LIN {X 0,Y 291.346,Z 740.192,A -85,B 0,C 180,E1 -16706.302,E2 -16706.302} C_VEL
LIN {X 0,Y 291.388,Z 740.187,A -85,B 0,C 180,E1 -16710.26,E2 -16710.26} C_VEL
LIN {X 0,Y 291.418,Z 740.184,A -85,B 0,C 180,E1 -16714.272,E2 -16714.272} C_VEL
LIN {X 0,Y 291.376,Z 740.187,A -85,B 0,C 180,E1 -16717.299,E2 -16717.299} C_VEL
LIN {X 0,Y 291.459,Z 740.18,A -85,B 0,C 180,E1 -16720.27,E2 -16720.27} C_VEL
LIN {X 0,Y 291.557,Z 740.166,A -85,B 0,C 180,E1 -16724.624,E2 -16724.624} C_VEL
LIN {X 0,Y 291.537,Z 740.167,A -85,B 0,C 180,E1 -16728.881,E2 -16728.881} C_VEL
LIN {X 0,Y 291.689,Z 740.147,A -85,B 0,C 180,E1 -16731.688,E2 -16731.688} C_VEL
LIN {X 0,Y 291.624,Z 740.161,A -85,B 0,C 180,E1 -16734.468,E2 -16734.468} C_VEL
LIN {X 0,Y 291.887,Z 740.128,A -85,B 0,C 180,E1 -16738.62,E2 -16738.62} C_VEL
LIN {X 0,Y 291.887,Z 740.123,A -85,B 0,C 180,E1 -16741.38,E2 -16741.38} C_VEL
LIN {X 0,Y 291.656,Z 740.153,A -85,B 0,C 180,E1 -16746.558,E2 -16746.558} C_VEL
LIN {X 0,Y 291.57,Z 740.163,A -85,B 0,C 180,E1 -16749.714,E2 -16749.714} C_VEL
LIN {X 0,Y 291.517,Z 740.169,A -85,B 0,C 180,E1 -16753.951,E2 -16753.951} C_VEL
LIN {X 0,Y 291.441,Z 740.178,A -85,B 0,C 180,E1 -16758.27,E2 -16758.27} C_VEL
LIN {X 0,Y 291.352,Z 740.195,A -85,B 0,C 180,E1 -16761.213,E2 -16761.213} C_VEL
LIN {X 0,Y 291.329,Z 740.192,A -85,B 0,C 180,E1 -16764.212,E2 -16764.212} C_VEL
LIN {X 0,Y 291.352,Z 740.193,A -85,B 0,C 180,E1 -16767.279,E2 -16767.279} C_VEL
LIN {X 0,Y 291.32,Z 740.194,A -85,B 0,C 180,E1 -16770.439,E2 -16770.439} C_VEL
LIN {X 0,Y 291.345,Z 740.195,A -85,B 0,C 180,E1 -16773.699,E2 -16773.699} C_VEL
LIN {X 0,Y 291.354,Z 740.191,A -85,B 0,C 180,E1 -16777.248,E2 -16777.248} C_VEL
LIN {X 0,Y 291.296,Z 740.2,A -85,B 0,C 180,E1 -16781.589,E2 -16781.589} C_VEL
LIN {X 0,Y 291.283,Z 740.201,A -85,B 0,C 180,E1 -16785.597,E2 -16785.597} C_VEL
LIN {X 0,Y 291.295,Z 740.197,A -85,B 0,C 180,E1 -16789.351,E2 -16789.351} C_VEL
LIN {X 0,Y 291.387,Z 740.185,A -85,B 0,C 180,E1 -16792.916,E2 -16792.916} C_VEL
LIN {X 0,Y 291.345,Z 740.195,A -85,B 0,C 180,E1 -16796.302,E2 -16796.302} C_VEL
LIN {X 0,Y 291.336,Z 740.196,A -85,B 0,C 180,E1 -16800.279,E2 -16800.279} C_VEL
LIN {X 0,Y 291.344,Z 740.195,A -85,B 0,C 180,E1 -16804.265,E2 -16804.265} C_VEL
LIN {X 0,Y 291.353,Z 740.189,A -85,B 0,C 180,E1 -16807.297,E2 -16807.297} C_VEL
LIN {X 0,Y 291.442,Z 740.18,A -85,B 0,C 180,E1 -16810.269,E2 -16810.269} C_VEL
LIN {X 0,Y 291.5,Z 740.176,A -85,B 0,C 180,E1 -16814.665,E2 -16814.665} C_VEL
LIN {X 0,Y 291.53,Z 740.173,A -85,B 0,C 180,E1 -16818.88,E2 -16818.88} C_VEL
LIN {X 0,Y 291.653,Z 740.152,A -85,B 0,C 180,E1 -16821.687,E2 -16821.687} C_VEL
LIN {X 0,Y 291.598,Z 740.16,A -85,B 0,C 180,E1 -16824.468,E2 -16824.468} C_VEL
LIN {X 0,Y 291.879,Z 740.125,A -85,B 0,C 180,E1 -16828.62,E2 -16828.62} C_VEL
LIN {X 0,Y 291.873,Z 740.128,A -85,B 0,C 180,E1 -16831.38,E2 -16831.38} C_VEL
LIN {X 0,Y 291.69,Z 740.149,A -85,B 0,C 180,E1 -16836.919,E2 -16836.919} C_VEL
LIN {X 0,Y 291.571,Z 740.165,A -85,B 0,C 180,E1 -16839.714,E2 -16839.714} C_VEL
LIN {X 0,Y 291.525,Z 740.17,A -85,B 0,C 180,E1 -16843.95,E2 -16843.95} C_VEL
LIN {X 0,Y 291.49,Z 740.173,A -85,B 0,C 180,E1 -16846.818,E2 -16846.818} C_VEL
LIN {X 0,Y 291.454,Z 740.18,A -85,B 0,C 180,E1 -16849.875,E2 -16849.875} C_VEL
LIN {X 0,Y 291.366,Z 740.19,A -85,B 0,C 180,E1 -16854.209,E2 -16854.209} C_VEL
LIN {X 0,Y 291.356,Z 740.19,A -85,B 0,C 180,E1 -16857.279,E2 -16857.279} C_VEL
LIN {X 0,Y 291.321,Z 740.196,A -85,B 0,C 180,E1 -16860.439,E2 -16860.439} C_VEL
LIN {X 0,Y 291.347,Z 740.193,A -85,B 0,C 180,E1 -16863.698,E2 -16863.698} C_VEL
LIN {X 0,Y 291.384,Z 740.186,A -85,B 0,C 180,E1 -16867.255,E2 -16867.255} C_VEL
LIN {X 0,Y 291.399,Z 740.188,A -85,B 0,C 180,E1 -16870.351,E2 -16870.351} C_VEL
LIN {X 0,Y 295.39,Z 753.65,A -85,B 0,C 180,E1 -16871.774,E2 -16871.774} C_VEL
LIN {X 0,Y 298.155,Z 764.257,A -85,B 0,C 180,E1 -16873.124,E2 -16873.124} C_VEL
LIN {X 0,Y 297.198,Z 775.278,A -85,B 0,C 180,E1 -16874.571,E2 -16874.571} C_VEL
LIN {X 0,Y 296.116,Z 785.835,A -85,B 0,C 180,E1 -16876.273,E2 -16876.273} C_VEL
LIN {X 0,Y 294.969,Z 795.249,A -85,B 0,C 180,E1 -16878.153,E2 -16878.153} C_VEL
LIN {X 0,Y 293.97,Z 803.803,A -85,B 0,C 180,E1 -16880.263,E2 -16880.263} C_VEL
LIN {X 0,Y 293.218,Z 810.365,A -85,B 0,C 180,E1 -16882.276,E2 -16882.276} C_VEL
LIN {X 0,Y 292.489,Z 816.762,A -85,B 0,C 180,E1 -16884.782,E2 -16884.782} C_VEL
LIN {X 0,Y 292.073,Z 821.66,A -85,B 0,C 180,E1 -16887.372,E2 -16887.372} C_VEL
LIN {X 0,Y 291.863,Z 825.094,A -85,B 0,C 180,E1 -16890.098,E2 -16890.098} C_VEL
LIN {X 0,Y 292.001,Z 826.918,A -85,B 0,C 180,E1 -16892.787,E2 -16892.787} C_VEL
LIN {X 0,Y 292.268,Z 827.255,A -85,B 0,C 180,E1 -16894.352,E2 -16894.352} C_VEL
LIN {X 0,Y 292.61,Z 827.12,A -85,B 0,C 180,E1 -16895.901,E2 -16895.901} C_VEL
LIN {X 0,Y 293.083,Z 826.429,A -85,B 0,C 180,E1 -16897.438,E2 -16897.438} C_VEL
LIN {X 0,Y 293.687,Z 825.284,A -85,B 0,C 180,E1 -16898.964,E2 -16898.964} C_VEL
LIN {X 0,Y 294.663,Z 822.645,A -85,B 0,C 180,E1 -16901.217,E2 -16901.217} C_VEL
LIN {X 0,Y 296.004,Z 818.763,A -85,B 0,C 180,E1 -16903.446,E2 -16903.446} C_VEL
LIN {X 0,Y 297.717,Z 813.148,A -85,B 0,C 180,E1 -16905.81,E2 -16905.81} C_VEL
LIN {X 0,Y 299.467,Z 806.982,A -85,B 0,C 180,E1 -16907.806,E2 -16907.806} C_VEL
LIN {X 0,Y 301.445,Z 798.721,A -85,B 0,C 180,E1 -16909.929,E2 -16909.929} C_VEL
LIN {X 0,Y 303.384,Z 790.165,A -85,B 0,C 180,E1 -16911.675,E2 -16911.675} C_VEL
LIN {X 0,Y 305.048,Z 781.584,A -85,B 0,C 180,E1 -16913.112,E2 -16913.112} C_VEL
LIN {X 0,Y 305.862,Z 775.886,A -85,B 0,C 180,E1 -16913.953,E2 -16913.953} C_VEL
LIN {X 0,Y 303.788,Z 767.821,A -85,B 0,C 180,E1 -16915.422,E2 -16915.422} C_VEL
LIN {X 0,Y 301.043,Z 760.013,A -85,B 0,C 180,E1 -16916.805,E2 -16916.805} C_VEL
LIN {X 0,Y 295.849,Z 748.049,A -85,B 0,C 180,E1 -16918.837,E2 -16918.837} C_VEL
LIN {X 0,Y 295.454,Z 747.403,A -85,B 0,C 180,E1 -16918.961,E2 -16918.961} C_VEL
LIN {X 0,Y 293.453,Z 745.045,A -85,B 0,C 180,E1 -16919.5,E2 -16919.5} C_VEL
LIN {X 0,Y 289.167,Z 742.472,A -85,B 0,C 180,E1 -16920.454,E2 -16920.454} C_VEL
LIN {X 0,Y 286.173,Z 741.381,A -85,B 0,C 180,E1 -16921.331,E2 -16921.331} C_VEL
LIN {X 0,Y 284.879,Z 741.031,A -85,B 0,C 180,E1 -16922.085,E2 -16922.085} C_VEL
LIN {X 0,Y 284.761,Z 741.007,A -85,B 0,C 180,E1 -16922.352,E2 -16922.352} C_VEL
LIN {X 0,Y 284.689,Z 741.021,A -85,B 0,C 180,E1 -16927.09,E2 -16927.09} C_VEL
LIN {X 0,Y 284.522,Z 741.039,A -85,B 0,C 180,E1 -16929.957,E2 -16929.957} C_VEL
LIN {X 0,Y 284.485,Z 741.043,A -85,B 0,C 180,E1 -16934.303,E2 -16934.303} C_VEL
LIN {X 0,Y 284.428,Z 741.052,A -85,B 0,C 180,E1 -16937.248,E2 -16937.248} C_VEL
LIN {X 0,Y 284.38,Z 741.058,A -85,B 0,C 180,E1 -16940.242,E2 -16940.242} C_VEL
LIN {X 0,Y 284.339,Z 741.065,A -85,B 0,C 180,E1 -16944.846,E2 -16944.846} C_VEL
LIN {X 0,Y 284.33,Z 741.067,A -85,B 0,C 180,E1 -16948.011,E2 -16948.011} C_VEL
LIN {X 0,Y 284.378,Z 741.283,A -85,B 0,C 180,E1 -16949.961,E2 -16949.961} C_VEL
LIN {X 0,Y 284.925,Z 743.801,A -85,B 0,C 180,E1 -16953.002,E2 -16953.002} C_VEL
LIN {X 0,Y 285.653,Z 746.974,A -85,B 0,C 180,E1 -16956.191,E2 -16956.191} C_VEL
LIN {X 0,Y 286.553,Z 750.978,A -85,B 0,C 180,E1 -16959.619,E2 -16959.619} C_VEL
LIN {X 0,Y 287.534,Z 755.832,A -85,B 0,C 180,E1 -16963.187,E2 -16963.187} C_VEL
LIN {X 0,Y 288.642,Z 761.7,A -85,B 0,C 180,E1 -16966.925,E2 -16966.925} C_VEL
LIN {X 0,Y 289.605,Z 767.03,A -85,B 0,C 180,E1 -16969.978,E2 -16969.978} C_VEL
LIN {X 0,Y 289.804,Z 768.763,A -85,B 0,C 180,E1 -16970.911,E2 -16970.911} C_VEL
LIN {X 0,Y 288.885,Z 773.995,A -85,B 0,C 180,E1 -16973.401,E2 -16973.401} C_VEL
LIN {X 0,Y 287.081,Z 782.923,A -85,B 0,C 180,E1 -16977.413,E2 -16977.413} C_VEL
LIN {X 0,Y 286.057,Z 790.173,A -85,B 0,C 180,E1 -16980.457,E2 -16980.457} C_VEL
LIN {X 0,Y 286.958,Z 794.013,A -85,B 0,C 180,E1 -16980.809,E2 -16980.809} C_VEL
LIN {X 0,Y 289.321,Z 804.43,A -85,B 0,C 180,E1 -16981.849,E2 -16981.849} C_VEL
LIN {X 0,Y 291.377,Z 817.452,A -85,B 0,C 180,E1 -16983.181,E2 -16983.181} C_VEL
LIN {X 0,Y 292.203,Z 829.766,A -85,B 0,C 180,E1 -16984.537,E2 -16984.537} C_VEL
LIN {X 0,Y 292.108,Z 840.627,A -85,B 0,C 180,E1 -16985.857,E2 -16985.857} C_VEL
LIN {X 0,Y 291.086,Z 852.313,A -85,B 0,C 180,E1 -16987.462,E2 -16987.462} C_VEL
LIN {X 0,Y 290.017,Z 862.075,A -85,B 0,C 180,E1 -16989.057,E2 -16989.057} C_VEL
LIN {X 0,Y 289.18,Z 867.757,A -85,B 0,C 180,E1 -16990.108,E2 -16990.108} C_VEL
LIN {X 0,Y 286.894,Z 877.547,A -85,B 0,C 180,E1 -16992.169,E2 -16992.169} C_VEL
LIN {X 0,Y 285.252,Z 885.594,A -85,B 0,C 180,E1 -16994.275,E2 -16994.275} C_VEL
LIN {X 0,Y 284.228,Z 892.25,A -85,B 0,C 180,E1 -16996.414,E2 -16996.414} C_VEL
LIN {X 0,Y 283.489,Z 897.677,A -85,B 0,C 180,E1 -16998.561,E2 -16998.561} C_VEL
LIN {X 0,Y 283.215,Z 902.021,A -85,B 0,C 180,E1 -17000.718,E2 -17000.718} C_VEL
LIN {X 0,Y 283.239,Z 905.511,A -85,B 0,C 180,E1 -17002.988,E2 -17002.988} C_VEL
LIN {X 0,Y 283.617,Z 908.327,A -85,B 0,C 180,E1 -17005.737,E2 -17005.737} C_VEL
LIN {X 0,Y 283.773,Z 909.165,A -85,B 0,C 180,E1 -17007.161,E2 -17007.161} C_VEL
LIN {X 0,Y 283.935,Z 909.542,A -85,B 0,C 180,E1 -17008.582,E2 -17008.582} C_VEL
LIN {X 0,Y 284.199,Z 909.518,A -85,B 0,C 180,E1 -17010,E2 -17010} C_VEL
LIN {X 0,Y 284.012,Z 909.006,A -85,B 0,C 180,E1 -17011.418,E2 -17011.418} C_VEL
LIN {X 0,Y 283.895,Z 908.063,A -85,B 0,C 180,E1 -17012.838,E2 -17012.838} C_VEL
LIN {X 0,Y 283.788,Z 906.629,A -85,B 0,C 180,E1 -17014.261,E2 -17014.261} C_VEL
LIN {X 0,Y 283.582,Z 903.606,A -85,B 0,C 180,E1 -17016.403,E2 -17016.403} C_VEL
LIN {X 0,Y 283.483,Z 899.442,A -85,B 0,C 180,E1 -17018.554,E2 -17018.554} C_VEL
LIN {X 0,Y 283.675,Z 893.034,A -85,B 0,C 180,E1 -17021.07,E2 -17021.07} C_VEL
LIN {X 0,Y 284.245,Z 886.007,A -85,B 0,C 180,E1 -17023.221,E2 -17023.221} C_VEL
LIN {X 0,Y 285.215,Z 877.236,A -85,B 0,C 180,E1 -17025.36,E2 -17025.36} C_VEL
LIN {X 0,Y 286.444,Z 867.317,A -85,B 0,C 180,E1 -17027.307,E2 -17027.307} C_VEL
LIN {X 0,Y 287.546,Z 858.519,A -85,B 0,C 180,E1 -17028.711,E2 -17028.711} C_VEL
LIN {X 0,Y 287.331,Z 847.324,A -85,B 0,C 180,E1 -17030.205,E2 -17030.205} C_VEL
LIN {X 0,Y 286.963,Z 834.809,A -85,B 0,C 180,E1 -17031.553,E2 -17031.553} C_VEL
LIN {X 0,Y 286.091,Z 821.64,A -85,B 0,C 180,E1 -17032.667,E2 -17032.667} C_VEL
LIN {X 0,Y 284.91,Z 807.176,A -85,B 0,C 180,E1 -17033.568,E2 -17033.568} C_VEL
LIN {X 0,Y 284.391,Z 801.447,A -85,B 0,C 180,E1 -17033.885,E2 -17033.885} C_VEL
LIN {X 0,Y 285.455,Z 791.716,A -85,B 0,C 180,E1 -17037.891,E2 -17037.891} C_VEL
LIN {X 0,Y 286.689,Z 782.298,A -85,B 0,C 180,E1 -17041.807,E2 -17041.807} C_VEL
LIN {X 0,Y 288.579,Z 771.122,A -85,B 0,C 180,E1 -17046.517,E2 -17046.517} C_VEL
LIN {X 0,Y 289.217,Z 767.266,A -85,B 0,C 180,E1 -17048.16,E2 -17048.16} C_VEL
LIN {X 0,Y 288.67,Z 763.06,A -85,B 0,C 180,E1 -17050.061,E2 -17050.061} C_VEL
LIN {X 0,Y 287.039,Z 754.864,A -85,B 0,C 180,E1 -17053.961,E2 -17053.961} C_VEL
LIN {X 0,Y 285.31,Z 746.209,A -85,B 0,C 180,E1 -17058.311,E2 -17058.311} C_VEL
LIN {X 0,Y 284.34,Z 741.066,A -85,B 0,C 180,E1 -17061.043,E2 -17061.043} C_VEL
LIN {X 0,Y 284.342,Z 741.063,A -85,B 0,C 180,E1 -17064.652,E2 -17064.652} C_VEL
LIN {X 0,Y 284.297,Z 741.069,A -85,B 0,C 180,E1 -17068.726,E2 -17068.726} C_VEL
LIN {X 0,Y 284.398,Z 741.055,A -85,B 0,C 180,E1 -17072.826,E2 -17072.826} C_VEL
LIN {X 0,Y 284.335,Z 741.064,A -85,B 0,C 180,E1 -17076.704,E2 -17076.704} C_VEL
LIN {X 0,Y 284.404,Z 741.054,A -85,B 0,C 180,E1 -17081.262,E2 -17081.262} C_VEL
LIN {X 0,Y 284.494,Z 741.047,A -85,B 0,C 180,E1 -17084.459,E2 -17084.459} C_VEL
LIN {X 0,Y 284.489,Z 741.047,A -85,B 0,C 180,E1 -17088.602,E2 -17088.602} C_VEL
LIN {X 0,Y 284.641,Z 741.025,A -85,B 0,C 180,E1 -17091.481,E2 -17091.481} C_VEL
LIN {X 0,Y 284.595,Z 741.035,A -85,B 0,C 180,E1 -17094.331,E2 -17094.331} C_VEL
LIN {X 0,Y 284.853,Z 741.004,A -85,B 0,C 180,E1 -17098.586,E2 -17098.586} C_VEL
LIN {X 0,Y 284.853,Z 741,A -85,B 0,C 180,E1 -17101.414,E2 -17101.414} C_VEL
LIN {X 0,Y 284.649,Z 741.027,A -85,B 0,C 180,E1 -17107.091,E2 -17107.091} C_VEL
LIN {X 0,Y 284.516,Z 741.041,A -85,B 0,C 180,E1 -17109.957,E2 -17109.957} C_VEL
LIN {X 0,Y 284.465,Z 741.048,A -85,B 0,C 180,E1 -17114.304,E2 -17114.304} C_VEL
LIN {X 0,Y 284.376,Z 741.06,A -85,B 0,C 180,E1 -17118.741,E2 -17118.741} C_VEL
LIN {X 0,Y 284.304,Z 741.069,A -85,B 0,C 180,E1 -17121.765,E2 -17121.765} C_VEL
LIN {X 0,Y 284.286,Z 741.07,A -85,B 0,C 180,E1 -17124.852,E2 -17124.852} C_VEL
LIN {X 0,Y 284.283,Z 741.071,A -85,B 0,C 180,E1 -17128.016,E2 -17128.016} C_VEL
LIN {X 0,Y 284.286,Z 741.073,A -85,B 0,C 180,E1 -17131.276,E2 -17131.276} C_VEL
LIN {X 0,Y 284.337,Z 741.065,A -85,B 0,C 180,E1 -17135.347,E2 -17135.347} C_VEL
LIN {X 0,Y 284.264,Z 741.074,A -85,B 0,C 180,E1 -17138.177,E2 -17138.177} C_VEL
LIN {X 0,Y 284.238,Z 741.078,A -85,B 0,C 180,E1 -17142.117,E2 -17142.117} C_VEL
LIN {X 0,Y 284.239,Z 741.079,A -85,B 0,C 180,E1 -17146.186,E2 -17146.186} C_VEL
LIN {X 0,Y 284.256,Z 741.078,A -85,B 0,C 180,E1 -17150.037,E2 -17150.037} C_VEL
LIN {X 0,Y 284.319,Z 741.067,A -85,B 0,C 180,E1 -17153.612,E2 -17153.612} C_VEL
LIN {X 0,Y 284.307,Z 741.067,A -85,B 0,C 180,E1 -17157.191,E2 -17157.191} C_VEL
LIN {X 0,Y 284.311,Z 741.071,A -85,B 0,C 180,E1 -17160.371,E2 -17160.371} C_VEL
LIN {X 0,Y 284.297,Z 741.069,A -85,B 0,C 180,E1 -17163.579,E2 -17163.579} C_VEL
LIN {X 0,Y 284.31,Z 741.07,A -85,B 0,C 180,E1 -17166.702,E2 -17166.702} C_VEL
LIN {X 0,Y 284.378,Z 741.058,A -85,B 0,C 180,E1 -17169.905,E2 -17169.905} C_VEL
LIN {X 0,Y 284.449,Z 741.053,A -85,B 0,C 180,E1 -17174.493,E2 -17174.493} C_VEL
LIN {X 0,Y 284.468,Z 741.05,A -85,B 0,C 180,E1 -17178.601,E2 -17178.601} C_VEL
LIN {X 0,Y 284.61,Z 741.031,A -85,B 0,C 180,E1 -17181.48,E2 -17181.48} C_VEL
LIN {X 0,Y 284.569,Z 741.035,A -85,B 0,C 180,E1 -17184.331,E2 -17184.331} C_VEL
LIN {X 0,Y 284.845,Z 741.001,A -85,B 0,C 180,E1 -17188.586,E2 -17188.586} C_VEL
LIN {X 0,Y 284.84,Z 741.004,A -85,B 0,C 180,E1 -17191.414,E2 -17191.414} C_VEL
LIN {X 0,Y 284.645,Z 741.028,A -85,B 0,C 180,E1 -17197.092,E2 -17197.092} C_VEL
LIN {X 0,Y 284.517,Z 741.042,A -85,B 0,C 180,E1 -17199.957,E2 -17199.957} C_VEL
LIN {X 0,Y 284.485,Z 741.045,A -85,B 0,C 180,E1 -17204.303,E2 -17204.303} C_VEL
LIN {X 0,Y 284.426,Z 741.055,A -85,B 0,C 180,E1 -17207.249,E2 -17207.249} C_VEL
LIN {X 0,Y 284.38,Z 741.059,A -85,B 0,C 180,E1 -17210.242,E2 -17210.242} C_VEL
LIN {X 0,Y 284.326,Z 741.07,A -85,B 0,C 180,E1 -17213.854,E2 -17213.854} C_VEL
LIN {X 0,Y 284.286,Z 741.075,A -85,B 0,C 180,E1 -17218.016,E2 -17218.016} C_VEL
LIN {X 0,Y 284.288,Z 741.07,A -85,B 0,C 180,E1 -17221.276,E2 -17221.276} C_VEL
LIN {X 0,Y 284.344,Z 741.063,A -85,B 0,C 180,E1 -17225.348,E2 -17225.348} C_VEL
LIN {X 0,Y 284.339,Z 741.064,A -85,B 0,C 180,E1 -17229.529,E2 -17229.529} C_VEL
LIN {X 0,Y 284.354,Z 741.136,A -85,B 0,C 180,E1 -17229.987,E2 -17229.987} C_VEL
LIN {X 0,Y 288.303,Z 754.235,A -85,B 0,C 180,E1 -17231.394,E2 -17231.394} C_VEL
LIN {X 0,Y 291.105,Z 764.997,A -85,B 0,C 180,E1 -17232.783,E2 -17232.783} C_VEL
LIN {X 0,Y 291.038,Z 768.945,A -85,B 0,C 180,E1 -17233.288,E2 -17233.288} C_VEL
LIN {X 0,Y 290.014,Z 779.201,A -85,B 0,C 180,E1 -17234.756,E2 -17234.756} C_VEL
LIN {X 0,Y 288.795,Z 789.796,A -85,B 0,C 180,E1 -17236.617,E2 -17236.617} C_VEL
LIN {X 0,Y 287.651,Z 799.415,A -85,B 0,C 180,E1 -17238.725,E2 -17238.725} C_VEL
LIN {X 0,Y 286.684,Z 807.034,A -85,B 0,C 180,E1 -17240.792,E2 -17240.792} C_VEL
LIN {X 0,Y 285.893,Z 813.513,A -85,B 0,C 180,E1 -17242.967,E2 -17242.967} C_VEL
LIN {X 0,Y 285.319,Z 819.315,A -85,B 0,C 180,E1 -17245.49,E2 -17245.49} C_VEL
LIN {X 0,Y 284.986,Z 823.541,A -85,B 0,C 180,E1 -17247.98,E2 -17247.98} C_VEL
LIN {X 0,Y 284.836,Z 826.398,A -85,B 0,C 180,E1 -17250.43,E2 -17250.43} C_VEL
LIN {X 0,Y 284.974,Z 827.867,A -85,B 0,C 180,E1 -17252.603,E2 -17252.603} C_VEL
LIN {X 0,Y 285.457,Z 828.368,A -85,B 0,C 180,E1 -17255.257,E2 -17255.257} C_VEL
LIN {X 0,Y 285.871,Z 827.999,A -85,B 0,C 180,E1 -17256.836,E2 -17256.836} C_VEL
LIN {X 0,Y 286.599,Z 826.891,A -85,B 0,C 180,E1 -17258.724,E2 -17258.724} C_VEL
LIN {X 0,Y 287.844,Z 823.949,A -85,B 0,C 180,E1 -17261.493,E2 -17261.493} C_VEL
LIN {X 0,Y 289.244,Z 820.152,A -85,B 0,C 180,E1 -17263.774,E2 -17263.774} C_VEL
LIN {X 0,Y 290.91,Z 815.071,A -85,B 0,C 180,E1 -17266.02,E2 -17266.02} C_VEL
LIN {X 0,Y 292.905,Z 808.567,A -85,B 0,C 180,E1 -17268.232,E2 -17268.232} C_VEL
LIN {X 0,Y 294.71,Z 801.878,A -85,B 0,C 180,E1 -17270.048,E2 -17270.048} C_VEL
LIN {X 0,Y 296.678,Z 793.806,A -85,B 0,C 180,E1 -17271.828,E2 -17271.828} C_VEL
LIN {X 0,Y 298.793,Z 783.622,A -85,B 0,C 180,E1 -17273.627,E2 -17273.627} C_VEL
LIN {X 0,Y 299.627,Z 779.064,A -85,B 0,C 180,E1 -17274.32,E2 -17274.32} C_VEL
LIN {X 0,Y 298.213,Z 772.155,A -85,B 0,C 180,E1 -17275.641,E2 -17275.641} C_VEL
LIN {X 0,Y 295.539,Z 764.064,A -85,B 0,C 180,E1 -17277.17,E2 -17277.17} C_VEL
LIN {X 0,Y 290.736,Z 752.389,A -85,B 0,C 180,E1 -17279.307,E2 -17279.307} C_VEL
LIN {X 0,Y 287.252,Z 745.57,A -85,B 0,C 180,E1 -17280.556,E2 -17280.556} C_VEL
LIN {X 0,Y 285.285,Z 742.718,A -85,B 0,C 180,E1 -17281.169,E2 -17281.169} C_VEL
LIN {X 0,Y 284.856,Z 741.003,A -85,B 0,C 180,E1 -17281.414,E2 -17281.414} C_VEL
LIN {X 0,Y 284.761,Z 741.007,A -85,B 0,C 180,E1 -17282.352,E2 -17282.352} C_VEL
LIN {X 0,Y 284.038,Z 741.099,A -85,B 0,C 180,E1 -17283.531,E2 -17283.531} C_VEL
LIN {X 0,Y 281.123,Z 741.46,A -85,B 0,C 180,E1 -17285.45,E2 -17285.45} C_VEL
LIN {X 0,Y 278.692,Z 741.767,A -85,B 0,C 180,E1 -17287.008,E2 -17287.008} C_VEL
LIN {X 0,Y 277.671,Z 741.891,A -85,B 0,C 180,E1 -17288.217,E2 -17288.217} C_VEL
LIN {X 0,Y 277.598,Z 741.897,A -85,B 0,C 180,E1 -17288.627,E2 -17288.627} C_VEL
LIN {X 0,Y 277.421,Z 741.926,A -85,B 0,C 180,E1 -17293.179,E2 -17293.179} C_VEL
LIN {X 0,Y 277.409,Z 741.927,A -85,B 0,C 180,E1 -17296.181,E2 -17296.181} C_VEL
LIN {X 0,Y 277.347,Z 741.933,A -85,B 0,C 180,E1 -17300.349,E2 -17300.349} C_VEL
LIN {X 0,Y 277.294,Z 741.938,A -85,B 0,C 180,E1 -17304.157,E2 -17304.157} C_VEL
LIN {X 0,Y 277.328,Z 742.119,A -85,B 0,C 180,E1 -17307.804,E2 -17307.804} C_VEL
LIN {X 0,Y 278.021,Z 745.311,A -85,B 0,C 180,E1 -17312.063,E2 -17312.063} C_VEL
LIN {X 0,Y 278.947,Z 749.292,A -85,B 0,C 180,E1 -17316.27,E2 -17316.27} C_VEL
LIN {X 0,Y 279.853,Z 753.39,A -85,B 0,C 180,E1 -17319.821,E2 -17319.821} C_VEL
LIN {X 0,Y 280.822,Z 758.285,A -85,B 0,C 180,E1 -17323.467,E2 -17323.467} C_VEL
LIN {X 0,Y 281.837,Z 763.788,A -85,B 0,C 180,E1 -17327.032,E2 -17327.032} C_VEL
LIN {X 0,Y 282.645,Z 768.346,A -85,B 0,C 180,E1 -17329.722,E2 -17329.722} C_VEL
LIN {X 0,Y 282.854,Z 770.695,A -85,B 0,C 180,E1 -17331,E2 -17331} C_VEL
LIN {X 0,Y 281.541,Z 777.058,A -85,B 0,C 180,E1 -17334.082,E2 -17334.082} C_VEL
LIN {X 0,Y 279.395,Z 788.307,A -85,B 0,C 180,E1 -17339.206,E2 -17339.206} C_VEL
LIN {X 0,Y 280.368,Z 792.51,A -85,B 0,C 180,E1 -17339.636,E2 -17339.636} C_VEL
LIN {X 0,Y 283.503,Z 806.189,A -85,B 0,C 180,E1 -17341.102,E2 -17341.102} C_VEL
LIN {X 0,Y 285.351,Z 820.401,A -85,B 0,C 180,E1 -17342.69,E2 -17342.69} C_VEL
LIN {X 0,Y 285.882,Z 832.505,A -85,B 0,C 180,E1 -17344.128,E2 -17344.128} C_VEL
LIN {X 0,Y 285.553,Z 842.787,A -85,B 0,C 180,E1 -17345.482,E2 -17345.482} C_VEL
LIN {X 0,Y 284.221,Z 854.811,A -85,B 0,C 180,E1 -17347.271,E2 -17347.271} C_VEL
LIN {X 0,Y 282.854,Z 865.832,A -85,B 0,C 180,E1 -17349.264,E2 -17349.264} C_VEL
LIN {X 0,Y 280.453,Z 875.75,A -85,B 0,C 180,E1 -17351.367,E2 -17351.367} C_VEL
LIN {X 0,Y 278.804,Z 883.186,A -85,B 0,C 180,E1 -17353.314,E2 -17353.314} C_VEL
LIN {X 0,Y 278.188,Z 886.263,A -85,B 0,C 180,E1 -17354.241,E2 -17354.241} C_VEL
LIN {X 0,Y 276.967,Z 893.505,A -85,B 0,C 180,E1 -17356.798,E2 -17356.798} C_VEL
LIN {X 0,Y 276.306,Z 898.47,A -85,B 0,C 180,E1 -17359.002,E2 -17359.002} C_VEL
LIN {X 0,Y 276.116,Z 902.395,A -85,B 0,C 180,E1 -17361.215,E2 -17361.215} C_VEL
LIN {X 0,Y 276.17,Z 904.799,A -85,B 0,C 180,E1 -17362.969,E2 -17362.969} C_VEL
LIN {X 0,Y 276.538,Z 907.343,A -85,B 0,C 180,E1 -17365.627,E2 -17365.627} C_VEL
LIN {X 0,Y 276.725,Z 908.119,A -85,B 0,C 180,E1 -17367.088,E2 -17367.088} C_VEL
LIN {X 0,Y 276.903,Z 908.468,A -85,B 0,C 180,E1 -17368.545,E2 -17368.545} C_VEL
LIN {X 0,Y 277.184,Z 908.417,A -85,B 0,C 180,E1 -17370,E2 -17370} C_VEL
LIN {X 0,Y 276.987,Z 907.869,A -85,B 0,C 180,E1 -17371.454,E2 -17371.454} C_VEL
LIN {X 0,Y 276.867,Z 906.85,A -85,B 0,C 180,E1 -17372.91,E2 -17372.91} C_VEL
LIN {X 0,Y 276.751,Z 905.376,A -85,B 0,C 180,E1 -17374.369,E2 -17374.369} C_VEL
LIN {X 0,Y 276.543,Z 902.27,A -85,B 0,C 180,E1 -17376.567,E2 -17376.567} C_VEL
LIN {X 0,Y 276.444,Z 898.015,A -85,B 0,C 180,E1 -17378.774,E2 -17378.774} C_VEL
LIN {X 0,Y 276.599,Z 892.522,A -85,B 0,C 180,E1 -17380.986,E2 -17380.986} C_VEL
LIN {X 0,Y 277.148,Z 885.647,A -85,B 0,C 180,E1 -17383.192,E2 -17383.192} C_VEL
LIN {X 0,Y 277.92,Z 878.63,A -85,B 0,C 180,E1 -17385.023,E2 -17385.023} C_VEL
LIN {X 0,Y 279.156,Z 869.189,A -85,B 0,C 180,E1 -17387.027,E2 -17387.027} C_VEL
LIN {X 0,Y 280.441,Z 859.881,A -85,B 0,C 180,E1 -17388.634,E2 -17388.634} C_VEL
LIN {X 0,Y 280.29,Z 847.824,A -85,B 0,C 180,E1 -17390.359,E2 -17390.359} C_VEL
LIN {X 0,Y 279.971,Z 835.553,A -85,B 0,C 180,E1 -17391.752,E2 -17391.752} C_VEL
LIN {X 0,Y 279.145,Z 822.067,A -85,B 0,C 180,E1 -17392.97,E2 -17392.97} C_VEL
LIN {X 0,Y 278.09,Z 808.245,A -85,B 0,C 180,E1 -17393.888,E2 -17393.888} C_VEL
LIN {X 0,Y 277.376,Z 800.496,A -85,B 0,C 180,E1 -17394.323,E2 -17394.323} C_VEL
LIN {X 0,Y 278.591,Z 790.349,A -85,B 0,C 180,E1 -17398.64,E2 -17398.64} C_VEL
LIN {X 0,Y 280.204,Z 779.041,A -85,B 0,C 180,E1 -17403.49,E2 -17403.49} C_VEL
LIN {X 0,Y 281.999,Z 769.354,A -85,B 0,C 180,E1 -17407.692,E2 -17407.692} C_VEL
LIN {X 0,Y 282.152,Z 767.523,A -85,B 0,C 180,E1 -17408.515,E2 -17408.515} C_VEL
LIN {X 0,Y 281.128,Z 761.385,A -85,B 0,C 180,E1 -17411.412,E2 -17411.412} C_VEL
LIN {X 0,Y 279.553,Z 753.622,A -85,B 0,C 180,E1 -17415.257,E2 -17415.257} C_VEL
LIN {X 0,Y 278.037,Z 745.814,A -85,B 0,C 180,E1 -17419.316,E2 -17419.316} C_VEL
LIN {X 0,Y 277.299,Z 741.944,A -85,B 0,C 180,E1 -17421.456,E2 -17421.456} C_VEL
LIN {X 0,Y 277.285,Z 741.943,A -85,B 0,C 180,E1 -17424.342,E2 -17424.342} C_VEL
LIN {X 0,Y 277.246,Z 741.952,A -85,B 0,C 180,E1 -17427.837,E2 -17427.837} C_VEL
LIN {X 0,Y 277.291,Z 741.942,A -85,B 0,C 180,E1 -17431.213,E2 -17431.213} C_VEL
LIN {X 0,Y 277.311,Z 741.94,A -85,B 0,C 180,E1 -17434.479,E2 -17434.479} C_VEL
LIN {X 0,Y 277.271,Z 741.946,A -85,B 0,C 180,E1 -17437.654,E2 -17437.654} C_VEL
LIN {X 0,Y 277.346,Z 741.934,A -85,B 0,C 180,E1 -17440.766,E2 -17440.766} C_VEL
LIN {X 0,Y 277.436,Z 741.923,A -85,B 0,C 180,E1 -17445.326,E2 -17445.326} C_VEL
LIN {X 0,Y 277.463,Z 741.92,A -85,B 0,C 180,E1 -17449.787,E2 -17449.787} C_VEL
LIN {X 0,Y 277.643,Z 741.901,A -85,B 0,C 180,E1 -17452.729,E2 -17452.729} C_VEL
LIN {X 0,Y 277.819,Z 741.88,A -85,B 0,C 180,E1 -17458.551,E2 -17458.551} C_VEL
LIN {X 0,Y 277.819,Z 741.876,A -85,B 0,C 180,E1 -17461.45,E2 -17461.45} C_VEL
LIN {X 0,Y 277.607,Z 741.902,A -85,B 0,C 180,E1 -17467.272,E2 -17467.272} C_VEL
LIN {X 0,Y 277.459,Z 741.92,A -85,B 0,C 180,E1 -17470.213,E2 -17470.213} C_VEL
LIN {X 0,Y 277.411,Z 741.928,A -85,B 0,C 180,E1 -17474.676,E2 -17474.676} C_VEL
LIN {X 0,Y 277.325,Z 741.942,A -85,B 0,C 180,E1 -17479.235,E2 -17479.235} C_VEL
LIN {X 0,Y 277.257,Z 741.945,A -85,B 0,C 180,E1 -17483.927,E2 -17483.927} C_VEL
LIN {X 0,Y 277.269,Z 741.949,A -85,B 0,C 180,E1 -17487.482,E2 -17487.482} C_VEL
LIN {X 0,Y 277.249,Z 741.946,A -85,B 0,C 180,E1 -17490.473,E2 -17490.473} C_VEL
LIN {X 0,Y 277.247,Z 741.949,A -85,B 0,C 180,E1 -17493.896,E2 -17493.896} C_VEL
LIN {X 0,Y 277.233,Z 741.952,A -85,B 0,C 180,E1 -17497.475,E2 -17497.475} C_VEL
LIN {X 0,Y 277.178,Z 741.956,A -85,B 0,C 180,E1 -17501.243,E2 -17501.243} C_VEL
LIN {X 0,Y 277.175,Z 741.956,A -85,B 0,C 180,E1 -17505.232,E2 -17505.232} C_VEL
LIN {X 0,Y 277.178,Z 741.955,A -85,B 0,C 180,E1 -17508.758,E2 -17508.758} C_VEL
LIN {X 0,Y 277.233,Z 741.95,A -85,B 0,C 180,E1 -17512.525,E2 -17512.525} C_VEL
LIN {X 0,Y 277.247,Z 741.951,A -85,B 0,C 180,E1 -17516.104,E2 -17516.104} C_VEL
LIN {X 0,Y 277.229,Z 741.948,A -85,B 0,C 180,E1 -17519.535,E2 -17519.535} C_VEL
LIN {X 0,Y 277.252,Z 741.948,A -85,B 0,C 180,E1 -17522.853,E2 -17522.853} C_VEL
LIN {X 0,Y 277.257,Z 741.947,A -85,B 0,C 180,E1 -17526.073,E2 -17526.073} C_VEL
LIN {X 0,Y 277.319,Z 741.942,A -85,B 0,C 180,E1 -17530.764,E2 -17530.764} C_VEL
LIN {X 0,Y 277.412,Z 741.926,A -85,B 0,C 180,E1 -17535.325,E2 -17535.325} C_VEL
LIN {X 0,Y 277.457,Z 741.921,A -85,B 0,C 180,E1 -17539.787,E2 -17539.787} C_VEL
LIN {X 0,Y 277.602,Z 741.906,A -85,B 0,C 180,E1 -17542.728,E2 -17542.728} C_VEL
LIN {X 0,Y 277.811,Z 741.877,A -85,B 0,C 180,E1 -17548.551,E2 -17548.551} C_VEL
LIN {X 0,Y 277.807,Z 741.88,A -85,B 0,C 180,E1 -17551.45,E2 -17551.45} C_VEL
LIN {X 0,Y 277.604,Z 741.906,A -85,B 0,C 180,E1 -17557.272,E2 -17557.272} C_VEL
LIN {X 0,Y 277.46,Z 741.92,A -85,B 0,C 180,E1 -17560.213,E2 -17560.213} C_VEL
LIN {X 0,Y 277.438,Z 741.922,A -85,B 0,C 180,E1 -17564.674,E2 -17564.674} C_VEL
LIN {X 0,Y 277.345,Z 741.936,A -85,B 0,C 180,E1 -17569.234,E2 -17569.234} C_VEL
LIN {X 0,Y 277.282,Z 741.945,A -85,B 0,C 180,E1 -17574.152,E2 -17574.152} C_VEL
LIN {X 0,Y 277.273,Z 741.946,A -85,B 0,C 180,E1 -17577.483,E2 -17577.483} C_VEL
LIN {X 0,Y 277.25,Z 741.948,A -85,B 0,C 180,E1 -17580.473,E2 -17580.473} C_VEL
LIN {X 0,Y 277.249,Z 741.951,A -85,B 0,C 180,E1 -17583.896,E2 -17583.896} C_VEL
LIN {X 0,Y 277.275,Z 741.944,A -85,B 0,C 180,E1 -17587.469,E2 -17587.469} C_VEL
LIN {X 0,Y 277.3,Z 741.941,A -85,B 0,C 180,E1 -17589.566,E2 -17589.566} C_VEL
LIN {X 0,Y 281.264,Z 755.199,A -85,B 0,C 180,E1 -17591.037,E2 -17591.037} C_VEL
LIN {X 0,Y 284.29,Z 766.808,A -85,B 0,C 180,E1 -17592.59,E2 -17592.59} C_VEL
LIN {X 0,Y 283.277,Z 778.606,A -85,B 0,C 180,E1 -17594.243,E2 -17594.243} C_VEL
LIN {X 0,Y 282.028,Z 789.299,A -85,B 0,C 180,E1 -17596.11,E2 -17596.11} C_VEL
LIN {X 0,Y 280.797,Z 799.254,A -85,B 0,C 180,E1 -17598.263,E2 -17598.263} C_VEL
LIN {X 0,Y 279.693,Z 807.87,A -85,B 0,C 180,E1 -17600.619,E2 -17600.619} C_VEL
LIN {X 0,Y 278.904,Z 814.234,A -85,B 0,C 180,E1 -17602.788,E2 -17602.788} C_VEL
LIN {X 0,Y 278.313,Z 820.152,A -85,B 0,C 180,E1 -17605.377,E2 -17605.377} C_VEL
LIN {X 0,Y 277.974,Z 824.44,A -85,B 0,C 180,E1 -17607.93,E2 -17607.93} C_VEL
LIN {X 0,Y 277.829,Z 826.548,A -85,B 0,C 180,E1 -17609.607,E2 -17609.607} C_VEL
LIN {X 0,Y 277.914,Z 828.681,A -85,B 0,C 180,E1 -17612.264,E2 -17612.264} C_VEL
LIN {X 0,Y 278.48,Z 829.508,A -85,B 0,C 180,E1 -17615.304,E2 -17615.304} C_VEL
LIN {X 0,Y 279.51,Z 828.447,A -85,B 0,C 180,E1 -17618.487,E2 -17618.487} C_VEL
LIN {X 0,Y 280.636,Z 826.212,A -85,B 0,C 180,E1 -17621,E2 -17621} C_VEL
LIN {X 0,Y 281.989,Z 822.917,A -85,B 0,C 180,E1 -17623.344,E2 -17623.344} C_VEL
LIN {X 0,Y 283.649,Z 818.387,A -85,B 0,C 180,E1 -17625.654,E2 -17625.654} C_VEL
LIN {X 0,Y 285.618,Z 812.502,A -85,B 0,C 180,E1 -17627.927,E2 -17627.927} C_VEL
LIN {X 0,Y 287.868,Z 805.004,A -85,B 0,C 180,E1 -17630.16,E2 -17630.16} C_VEL
LIN {X 0,Y 290.256,Z 796.028,A -85,B 0,C 180,E1 -17632.269,E2 -17632.269} C_VEL
LIN {X 0,Y 292.54,Z 785.979,A -85,B 0,C 180,E1 -17634.14,E2 -17634.14} C_VEL
LIN {X 0,Y 293.47,Z 781.043,A -85,B 0,C 180,E1 -17634.925,E2 -17634.925} C_VEL
LIN {X 0,Y 291.652,Z 773.019,A -85,B 0,C 180,E1 -17636.547,E2 -17636.547} C_VEL
LIN {X 0,Y 289.343,Z 766.23,A -85,B 0,C 180,E1 -17637.938,E2 -17637.938} C_VEL
LIN {X 0,Y 285.056,Z 755.611,A -85,B 0,C 180,E1 -17640,E2 -17640} C_VEL
LIN {X 0,Y 282.389,Z 750.296,A -85,B 0,C 180,E1 -17641.069,E2 -17641.069} C_VEL
LIN {X 0,Y 280.454,Z 746.999,A -85,B 0,C 180,E1 -17641.759,E2 -17641.759} C_VEL
LIN {X 0,Y 278.186,Z 743.633,A -85,B 0,C 180,E1 -17642.522,E2 -17642.522} C_VEL
LIN {X 0,Y 277.723,Z 741.883,A -85,B 0,C 180,E1 -17642.801,E2 -17642.801} C_VEL
LIN {X 0,Y 277.643,Z 741.9,A -85,B 0,C 180,E1 -17647.271,E2 -17647.271} C_VEL
LIN {X 0,Y 277.598,Z 741.897,A -85,B 0,C 180,E1 -17648.627,E2 -17648.627} C_VEL
LIN {X 0,Y 276.923,Z 741.987,A -85,B 0,C 180,E1 -17649.836,E2 -17649.836} C_VEL
LIN {X 0,Y 273.957,Z 742.351,A -85,B 0,C 180,E1 -17651.802,E2 -17651.802} C_VEL
LIN {X 0,Y 271.467,Z 742.67,A -85,B 0,C 180,E1 -17653.4,E2 -17653.4} C_VEL
LIN {X 0,Y 270.456,Z 742.788,A -85,B 0,C 180,E1 -17654.642,E2 -17654.642} C_VEL
LIN {X 0,Y 270.406,Z 742.793,A -85,B 0,C 180,E1 -17655.063,E2 -17655.063} C_VEL
LIN {X 0,Y 270.304,Z 742.816,A -85,B 0,C 180,E1 -17659.755,E2 -17659.755} C_VEL
LIN {X 0,Y 270.252,Z 742.82,A -85,B 0,C 180,E1 -17664.895,E2 -17664.895} C_VEL
LIN {X 0,Y 270.642,Z 744.59,A -85,B 0,C 180,E1 -17668.004,E2 -17668.004} C_VEL
LIN {X 0,Y 271.137,Z 746.914,A -85,B 0,C 180,E1 -17671.226,E2 -17671.226} C_VEL
LIN {X 0,Y 271.801,Z 749.95,A -85,B 0,C 180,E1 -17674.671,E2 -17674.671} C_VEL
LIN {X 0,Y 272.654,Z 753.652,A -85,B 0,C 180,E1 -17678.216,E2 -17678.216} C_VEL
LIN {X 0,Y 273.602,Z 758.211,A -85,B 0,C 180,E1 -17681.902,E2 -17681.902} C_VEL
LIN {X 0,Y 274.661,Z 763.714,A -85,B 0,C 180,E1 -17685.763,E2 -17685.763} C_VEL
LIN {X 0,Y 275.816,Z 770.357,A -85,B 0,C 180,E1 -17689.856,E2 -17689.856} C_VEL
LIN {X 0,Y 275.828,Z 773.155,A -85,B 0,C 180,E1 -17691.372,E2 -17691.372} C_VEL
LIN {X 0,Y 273.966,Z 780.955,A -85,B 0,C 180,E1 -17695.174,E2 -17695.174} C_VEL
LIN {X 0,Y 272.86,Z 786.921,A -85,B 0,C 180,E1 -17697.89,E2 -17697.89} C_VEL
LIN {X 0,Y 273.831,Z 790.934,A -85,B 0,C 180,E1 -17698.326,E2 -17698.326} C_VEL
LIN {X 0,Y 274.589,Z 793.745,A -85,B 0,C 180,E1 -17698.659,E2 -17698.659} C_VEL
LIN {X 0,Y 277.214,Z 805.811,A -85,B 0,C 180,E1 -17700.081,E2 -17700.081} C_VEL
LIN {X 0,Y 279.024,Z 819.128,A -85,B 0,C 180,E1 -17701.663,E2 -17701.663} C_VEL
LIN {X 0,Y 279.553,Z 830.483,A -85,B 0,C 180,E1 -17703.094,E2 -17703.094} C_VEL
LIN {X 0,Y 279.216,Z 841.993,A -85,B 0,C 180,E1 -17704.665,E2 -17704.665} C_VEL
LIN {X 0,Y 277.965,Z 852.918,A -85,B 0,C 180,E1 -17706.335,E2 -17706.335} C_VEL
LIN {X 0,Y 276.391,Z 863.942,A -85,B 0,C 180,E1 -17708.364,E2 -17708.364} C_VEL
LIN {X 0,Y 274.949,Z 870.841,A -85,B 0,C 180,E1 -17709.813,E2 -17709.813} C_VEL
LIN {X 0,Y 272.677,Z 879.597,A -85,B 0,C 180,E1 -17711.983,E2 -17711.983} C_VEL
LIN {X 0,Y 271.214,Z 885.752,A -85,B 0,C 180,E1 -17713.825,E2 -17713.825} C_VEL
LIN {X 0,Y 270.277,Z 890.992,A -85,B 0,C 180,E1 -17715.698,E2 -17715.698} C_VEL
LIN {X 0,Y 269.456,Z 896.201,A -85,B 0,C 180,E1 -17717.956,E2 -17717.956} C_VEL
LIN {X 0,Y 269.101,Z 900.373,A -85,B 0,C 180,E1 -17720.226,E2 -17720.226} C_VEL
LIN {X 0,Y 269.096,Z 904.099,A -85,B 0,C 180,E1 -17722.956,E2 -17722.956} C_VEL
LIN {X 0,Y 269.46,Z 906.337,A -85,B 0,C 180,E1 -17725.512,E2 -17725.512} C_VEL
LIN {X 0,Y 269.673,Z 907.073,A -85,B 0,C 180,E1 -17727.012,E2 -17727.012} C_VEL
LIN {X 0,Y 269.871,Z 907.395,A -85,B 0,C 180,E1 -17728.508,E2 -17728.508} C_VEL
LIN {X 0,Y 270.166,Z 907.317,A -85,B 0,C 180,E1 -17730,E2 -17730} C_VEL
LIN {X 0,Y 269.964,Z 906.708,A -85,B 0,C 180,E1 -17731.492,E2 -17731.492} C_VEL
LIN {X 0,Y 269.836,Z 905.639,A -85,B 0,C 180,E1 -17732.986,E2 -17732.986} C_VEL
LIN {X 0,Y 269.714,Z 904.129,A -85,B 0,C 180,E1 -17734.483,E2 -17734.483} C_VEL
LIN {X 0,Y 269.502,Z 900.939,A -85,B 0,C 180,E1 -17736.739,E2 -17736.739} C_VEL
LIN {X 0,Y 269.398,Z 896.592,A -85,B 0,C 180,E1 -17739.005,E2 -17739.005} C_VEL
LIN {X 0,Y 269.59,Z 891.004,A -85,B 0,C 180,E1 -17741.275,E2 -17741.275} C_VEL
LIN {X 0,Y 270.208,Z 883.994,A -85,B 0,C 180,E1 -17743.538,E2 -17743.538} C_VEL
LIN {X 0,Y 271.235,Z 875.238,A -85,B 0,C 180,E1 -17745.787,E2 -17745.787} C_VEL
LIN {X 0,Y 272.445,Z 866.024,A -85,B 0,C 180,E1 -17747.702,E2 -17747.702} C_VEL
LIN {X 0,Y 273.402,Z 858.864,A -85,B 0,C 180,E1 -17748.937,E2 -17748.937} C_VEL
LIN {X 0,Y 273.277,Z 846.811,A -85,B 0,C 180,E1 -17750.709,E2 -17750.709} C_VEL
LIN {X 0,Y 272.911,Z 834.607,A -85,B 0,C 180,E1 -17752.137,E2 -17752.137} C_VEL
LIN {X 0,Y 272.121,Z 821.059,A -85,B 0,C 180,E1 -17753.396,E2 -17753.396} C_VEL
LIN {X 0,Y 271.051,Z 807.413,A -85,B 0,C 180,E1 -17754.332,E2 -17754.332} C_VEL
LIN {X 0,Y 270.381,Z 799.626,A -85,B 0,C 180,E1 -17754.759,E2 -17754.759} C_VEL
LIN {X 0,Y 271.54,Z 790.386,A -85,B 0,C 180,E1 -17758.797,E2 -17758.797} C_VEL
LIN {X 0,Y 273.147,Z 779.537,A -85,B 0,C 180,E1 -17763.586,E2 -17763.586} C_VEL
LIN {X 0,Y 274.844,Z 770.651,A -85,B 0,C 180,E1 -17767.562,E2 -17767.562} C_VEL
LIN {X 0,Y 274.973,Z 766.995,A -85,B 0,C 180,E1 -17769.241,E2 -17769.241} C_VEL
LIN {X 0,Y 273.518,Z 759.539,A -85,B 0,C 180,E1 -17772.92,E2 -17772.92} C_VEL
LIN {X 0,Y 271.892,Z 751.619,A -85,B 0,C 180,E1 -17777.013,E2 -17777.013} C_VEL
LIN {X 0,Y 270.706,Z 745.223,A -85,B 0,C 180,E1 -17780.502,E2 -17780.502} C_VEL
LIN {X 0,Y 270.23,Z 742.824,A -85,B 0,C 180,E1 -17781.853,E2 -17781.853} C_VEL
LIN {X 0,Y 270.203,Z 742.825,A -85,B 0,C 180,E1 -17785.095,E2 -17785.095} C_VEL
LIN {X 0,Y 270.201,Z 742.826,A -85,B 0,C 180,E1 -17789.131,E2 -17789.131} C_VEL
LIN {X 0,Y 270.266,Z 742.818,A -85,B 0,C 180,E1 -17792.146,E2 -17792.146} C_VEL
LIN {X 0,Y 270.239,Z 742.821,A -85,B 0,C 180,E1 -17795.537,E2 -17795.537} C_VEL
LIN {X 0,Y 270.303,Z 742.815,A -85,B 0,C 180,E1 -17800.245,E2 -17800.245} C_VEL
LIN {X 0,Y 270.405,Z 742.8,A -85,B 0,C 180,E1 -17804.936,E2 -17804.936} C_VEL
LIN {X 0,Y 270.415,Z 742.797,A -85,B 0,C 180,E1 -17809.518,E2 -17809.518} C_VEL
LIN {X 0,Y 270.6,Z 742.779,A -85,B 0,C 180,E1 -17812.539,E2 -17812.539} C_VEL
LIN {X 0,Y 270.784,Z 742.755,A -85,B 0,C 180,E1 -17818.513,E2 -17818.513} C_VEL
LIN {X 0,Y 270.785,Z 742.752,A -85,B 0,C 180,E1 -17821.487,E2 -17821.487} C_VEL
LIN {X 0,Y 270.568,Z 742.778,A -85,B 0,C 180,E1 -17827.463,E2 -17827.463} C_VEL
LIN {X 0,Y 270.411,Z 742.799,A -85,B 0,C 180,E1 -17830.482,E2 -17830.482} C_VEL
LIN {X 0,Y 270.379,Z 742.806,A -85,B 0,C 180,E1 -17835.066,E2 -17835.066} C_VEL
LIN {X 0,Y 270.262,Z 742.818,A -85,B 0,C 180,E1 -17839.759,E2 -17839.759} C_VEL
LIN {X 0,Y 270.179,Z 742.826,A -85,B 0,C 180,E1 -17844.595,E2 -17844.595} C_VEL
LIN {X 0,Y 270.198,Z 742.826,A -85,B 0,C 180,E1 -17847.917,E2 -17847.917} C_VEL
LIN {X 0,Y 270.175,Z 742.831,A -85,B 0,C 180,E1 -17851.35,E2 -17851.35} C_VEL
LIN {X 0,Y 270.199,Z 742.824,A -85,B 0,C 180,E1 -17854.906,E2 -17854.906} C_VEL
LIN {X 0,Y 270.169,Z 742.829,A -85,B 0,C 180,E1 -17858.703,E2 -17858.703} C_VEL
LIN {X 0,Y 270.149,Z 742.83,A -85,B 0,C 180,E1 -17863.245,E2 -17863.245} C_VEL
LIN {X 0,Y 270.152,Z 742.832,A -85,B 0,C 180,E1 -17867.438,E2 -17867.438} C_VEL
LIN {X 0,Y 270.153,Z 742.829,A -85,B 0,C 180,E1 -17871.365,E2 -17871.365} C_VEL
LIN {X 0,Y 270.199,Z 742.825,A -85,B 0,C 180,E1 -17875.094,E2 -17875.094} C_VEL
LIN {X 0,Y 270.172,Z 742.827,A -85,B 0,C 180,E1 -17879.141,E2 -17879.141} C_VEL
LIN {X 0,Y 270.189,Z 742.829,A -85,B 0,C 180,E1 -17882.177,E2 -17882.177} C_VEL
LIN {X 0,Y 270.183,Z 742.827,A -85,B 0,C 180,E1 -17885.564,E2 -17885.564} C_VEL
LIN {X 0,Y 270.259,Z 742.818,A -85,B 0,C 180,E1 -17890.241,E2 -17890.241} C_VEL
LIN {X 0,Y 270.371,Z 742.806,A -85,B 0,C 180,E1 -17894.934,E2 -17894.934} C_VEL
LIN {X 0,Y 270.409,Z 742.799,A -85,B 0,C 180,E1 -17899.518,E2 -17899.518} C_VEL
LIN {X 0,Y 270.564,Z 742.781,A -85,B 0,C 180,E1 -17902.538,E2 -17902.538} C_VEL
LIN {X 0,Y 270.776,Z 742.753,A -85,B 0,C 180,E1 -17908.513,E2 -17908.513} C_VEL
LIN {X 0,Y 270.773,Z 742.756,A -85,B 0,C 180,E1 -17911.487,E2 -17911.487} C_VEL
LIN {X 0,Y 270.565,Z 742.784,A -85,B 0,C 180,E1 -17917.463,E2 -17917.463} C_VEL
LIN {X 0,Y 270.413,Z 742.798,A -85,B 0,C 180,E1 -17920.482,E2 -17920.482} C_VEL
LIN {X 0,Y 270.406,Z 742.799,A -85,B 0,C 180,E1 -17925.065,E2 -17925.065} C_VEL
LIN {X 0,Y 270.303,Z 742.816,A -85,B 0,C 180,E1 -17929.756,E2 -17929.756} C_VEL
LIN {X 0,Y 270.228,Z 742.821,A -85,B 0,C 180,E1 -17934.59,E2 -17934.59} C_VEL
LIN {X 0,Y 270.202,Z 742.83,A -85,B 0,C 180,E1 -17937.917,E2 -17937.917} C_VEL
LIN {X 0,Y 270.176,Z 742.829,A -85,B 0,C 180,E1 -17941.35,E2 -17941.35} C_VEL
LIN {X 0,Y 270.205,Z 742.825,A -85,B 0,C 180,E1 -17944.905,E2 -17944.905} C_VEL
LIN {X 0,Y 270.254,Z 742.819,A -85,B 0,C 180,E1 -17949.156,E2 -17949.156} C_VEL
LIN {X 0,Y 273.987,Z 755.359,A -85,B 0,C 180,E1 -17950.567,E2 -17950.567} C_VEL
LIN {X 0,Y 276.992,Z 766.477,A -85,B 0,C 180,E1 -17952.065,E2 -17952.065} C_VEL
LIN {X 0,Y 277.445,Z 769.052,A -85,B 0,C 180,E1 -17952.444,E2 -17952.444} C_VEL
LIN {X 0,Y 276.286,Z 780.338,A -85,B 0,C 180,E1 -17954.084,E2 -17954.084} C_VEL
LIN {X 0,Y 275.007,Z 790.82,A -85,B 0,C 180,E1 -17955.98,E2 -17955.98} C_VEL
LIN {X 0,Y 273.8,Z 800.452,A -85,B 0,C 180,E1 -17958.135,E2 -17958.135} C_VEL
LIN {X 0,Y 272.726,Z 808.41,A -85,B 0,C 180,E1 -17960.354,E2 -17960.354} C_VEL
LIN {X 0,Y 271.927,Z 814.857,A -85,B 0,C 180,E1 -17962.579,E2 -17962.579} C_VEL
LIN {X 0,Y 271.3,Z 820.945,A -85,B 0,C 180,E1 -17965.256,E2 -17965.256} C_VEL
LIN {X 0,Y 270.949,Z 825.315,A -85,B 0,C 180,E1 -17967.877,E2 -17967.877} C_VEL
LIN {X 0,Y 270.799,Z 828.318,A -85,B 0,C 180,E1 -17970.455,E2 -17970.455} C_VEL
LIN {X 0,Y 270.89,Z 829.625,A -85,B 0,C 180,E1 -17972.16,E2 -17972.16} C_VEL
LIN {X 0,Y 271.372,Z 830.588,A -85,B 0,C 180,E1 -17975.018,E2 -17975.018} C_VEL
LIN {X 0,Y 272.017,Z 830.336,A -85,B 0,C 180,E1 -17977.198,E2 -17977.198} C_VEL
LIN {X 0,Y 272.648,Z 829.59,A -85,B 0,C 180,E1 -17978.846,E2 -17978.846} C_VEL
LIN {X 0,Y 273.99,Z 827.125,A -85,B 0,C 180,E1 -17981.637,E2 -17981.637} C_VEL
LIN {X 0,Y 275.8,Z 822.984,A -85,B 0,C 180,E1 -17984.481,E2 -17984.481} C_VEL
LIN {X 0,Y 277.658,Z 818.109,A -85,B 0,C 180,E1 -17986.832,E2 -17986.832} C_VEL
LIN {X 0,Y 280.071,Z 811.192,A -85,B 0,C 180,E1 -17989.341,E2 -17989.341} C_VEL
LIN {X 0,Y 282.279,Z 803.952,A -85,B 0,C 180,E1 -17991.409,E2 -17991.409} C_VEL
LIN {X 0,Y 284.551,Z 795.78,A -85,B 0,C 180,E1 -17993.262,E2 -17993.262} C_VEL
LIN {X 0,Y 286.868,Z 785.874,A -85,B 0,C 180,E1 -17995.081,E2 -17995.081} C_VEL
LIN {X 0,Y 287.329,Z 783.657,A -85,B 0,C 180,E1 -17995.44,E2 -17995.44} C_VEL
LIN {X 0,Y 285.971,Z 776.858,A -85,B 0,C 180,E1 -17996.915,E2 -17996.915} C_VEL
LIN {X 0,Y 282.999,Z 767.772,A -85,B 0,C 180,E1 -17998.864,E2 -17998.864} C_VEL
LIN {X 0,Y 280.279,Z 760.579,A -85,B 0,C 180,E1 -18000.359,E2 -18000.359} C_VEL
LIN {X 0,Y 277.865,Z 755.501,A -85,B 0,C 180,E1 -18001.449,E2 -18001.449} C_VEL
LIN {X 0,Y 274.628,Z 750.215,A -85,B 0,C 180,E1 -18002.714,E2 -18002.714} C_VEL
LIN {X 0,Y 272.995,Z 747.278,A -85,B 0,C 180,E1 -18003.367,E2 -18003.367} C_VEL
LIN {X 0,Y 271.141,Z 745.027,A -85,B 0,C 180,E1 -18003.994,E2 -18003.994} C_VEL
LIN {X 0,Y 270.431,Z 742.8,A -85,B 0,C 180,E1 -18004.378,E2 -18004.378} C_VEL
LIN {X 0,Y 270.601,Z 742.778,A -85,B 0,C 180,E1 -18007.461,E2 -18007.461} C_VEL
LIN {X 0,Y 270.416,Z 742.802,A -85,B 0,C 180,E1 -18010.482,E2 -18010.482} C_VEL
LIN {X 0,Y 270.406,Z 742.793,A -85,B 0,C 180,E1 -18015.063,E2 -18015.063} C_VEL
LIN {X 0,Y 269.793,Z 742.896,A -85,B 0,C 180,E1 -18016.306,E2 -18016.306} C_VEL
LIN {X 0,Y 266.847,Z 743.237,A -85,B 0,C 180,E1 -18018.327,E2 -18018.327} C_VEL
LIN {X 0,Y 264.312,Z 743.56,A -85,B 0,C 180,E1 -18019.97,E2 -18019.97} C_VEL
LIN {X 0,Y 263.239,Z 743.687,A -85,B 0,C 180,E1 -18021.246,E2 -18021.246} C_VEL
LIN {X 0,Y 263.163,Z 743.764,A -85,B 0,C 180,E1 -18021.677,E2 -18021.677} C_VEL
LIN {X 0,Y 263.591,Z 745.34,A -85,B 0,C 180,E1 -18025.252,E2 -18025.252} C_VEL
LIN {X 0,Y 264.005,Z 747.354,A -85,B 0,C 180,E1 -18028.631,E2 -18028.631} C_VEL
LIN {X 0,Y 264.585,Z 749.948,A -85,B 0,C 180,E1 -18032.09,E2 -18032.09} C_VEL
LIN {X 0,Y 265.281,Z 753.17,A -85,B 0,C 180,E1 -18035.65,E2 -18035.65} C_VEL
LIN {X 0,Y 266.215,Z 757.093,A -85,B 0,C 180,E1 -18039.316,E2 -18039.316} C_VEL
LIN {X 0,Y 267.157,Z 761.958,A -85,B 0,C 180,E1 -18043.155,E2 -18043.155} C_VEL
LIN {X 0,Y 268.196,Z 767.617,A -85,B 0,C 180,E1 -18047.052,E2 -18047.052} C_VEL
LIN {X 0,Y 269,Z 772.839,A -85,B 0,C 180,E1 -18050.26,E2 -18050.26} C_VEL
LIN {X 0,Y 268.662,Z 775.527,A -85,B 0,C 180,E1 -18051.7,E2 -18051.7} C_VEL
LIN {X 0,Y 266.765,Z 783.136,A -85,B 0,C 180,E1 -18055.498,E2 -18055.498} C_VEL
LIN {X 0,Y 266.382,Z 785.182,A -85,B 0,C 180,E1 -18056.406,E2 -18056.406} C_VEL
LIN {X 0,Y 267.395,Z 789.305,A -85,B 0,C 180,E1 -18056.908,E2 -18056.908} C_VEL
LIN {X 0,Y 268.145,Z 792.052,A -85,B 0,C 180,E1 -18057.272,E2 -18057.272} C_VEL
LIN {X 0,Y 270.752,Z 803.465,A -85,B 0,C 180,E1 -18058.725,E2 -18058.725} C_VEL
LIN {X 0,Y 272.582,Z 816.111,A -85,B 0,C 180,E1 -18060.344,E2 -18060.344} C_VEL
LIN {X 0,Y 273.335,Z 828.013,A -85,B 0,C 180,E1 -18061.914,E2 -18061.914} C_VEL
LIN {X 0,Y 273.068,Z 840.139,A -85,B 0,C 180,E1 -18063.642,E2 -18063.642} C_VEL
LIN {X 0,Y 271.668,Z 852.143,A -85,B 0,C 180,E1 -18065.549,E2 -18065.549} C_VEL
LIN {X 0,Y 269.975,Z 862.181,A -85,B 0,C 180,E1 -18067.42,E2 -18067.42} C_VEL
LIN {X 0,Y 268.74,Z 869.115,A -85,B 0,C 180,E1 -18068.925,E2 -18068.925} C_VEL
LIN {X 0,Y 266.24,Z 877.919,A -85,B 0,C 180,E1 -18071.133,E2 -18071.133} C_VEL
LIN {X 0,Y 264.153,Z 886.332,A -85,B 0,C 180,E1 -18073.778,E2 -18073.778} C_VEL
LIN {X 0,Y 263.018,Z 892.203,A -85,B 0,C 180,E1 -18076.085,E2 -18076.085} C_VEL
LIN {X 0,Y 262.265,Z 896.945,A -85,B 0,C 180,E1 -18078.406,E2 -18078.406} C_VEL
LIN {X 0,Y 261.988,Z 900.677,A -85,B 0,C 180,E1 -18080.738,E2 -18080.738} C_VEL
LIN {X 0,Y 262.04,Z 903.305,A -85,B 0,C 180,E1 -18082.911,E2 -18082.911} C_VEL
LIN {X 0,Y 262.385,Z 905.321,A -85,B 0,C 180,E1 -18085.391,E2 -18085.391} C_VEL
LIN {X 0,Y 262.618,Z 906.025,A -85,B 0,C 180,E1 -18086.932,E2 -18086.932} C_VEL
LIN {X 0,Y 262.837,Z 906.314,A -85,B 0,C 180,E1 -18088.468,E2 -18088.468} C_VEL
LIN {X 0,Y 263.173,Z 906.194,A -85,B 0,C 180,E1 -18090,E2 -18090} C_VEL
LIN {X 0,Y 262.968,Z 905.513,A -85,B 0,C 180,E1 -18091.531,E2 -18091.531} C_VEL
LIN {X 0,Y 262.806,Z 904.402,A -85,B 0,C 180,E1 -18093.066,E2 -18093.066} C_VEL
LIN {X 0,Y 262.613,Z 901.874,A -85,B 0,C 180,E1 -18095.374,E2 -18095.374} C_VEL
LIN {X 0,Y 262.4,Z 898.215,A -85,B 0,C 180,E1 -18097.696,E2 -18097.696} C_VEL
LIN {X 0,Y 262.413,Z 893.368,A -85,B 0,C 180,E1 -18100.025,E2 -18100.025} C_VEL
LIN {X 0,Y 262.816,Z 887.229,A -85,B 0,C 180,E1 -18102.353,E2 -18102.353} C_VEL
LIN {X 0,Y 263.585,Z 879.547,A -85,B 0,C 180,E1 -18104.673,E2 -18104.673} C_VEL
LIN {X 0,Y 264.844,Z 869.966,A -85,B 0,C 180,E1 -18106.972,E2 -18106.972} C_VEL
LIN {X 0,Y 266.277,Z 860.156,A -85,B 0,C 180,E1 -18108.864,E2 -18108.864} C_VEL
LIN {X 0,Y 266.218,Z 848.586,A -85,B 0,C 180,E1 -18110.676,E2 -18110.676} C_VEL
LIN {X 0,Y 265.956,Z 836.028,A -85,B 0,C 180,E1 -18112.267,E2 -18112.267} C_VEL
LIN {X 0,Y 265.231,Z 822.58,A -85,B 0,C 180,E1 -18113.598,E2 -18113.598} C_VEL
LIN {X 0,Y 264.233,Z 808.856,A -85,B 0,C 180,E1 -18114.634,E2 -18114.634} C_VEL
LIN {X 0,Y 263.371,Z 798.718,A -85,B 0,C 180,E1 -18115.201,E2 -18115.201} C_VEL
LIN {X 0,Y 264.618,Z 789.374,A -85,B 0,C 180,E1 -18119.428,E2 -18119.428} C_VEL
LIN {X 0,Y 266.4,Z 778.305,A -85,B 0,C 180,E1 -18124.468,E2 -18124.468} C_VEL
LIN {X 0,Y 267.958,Z 770.382,A -85,B 0,C 180,E1 -18128.109,E2 -18128.109} C_VEL
LIN {X 0,Y 267.794,Z 767.134,A -85,B 0,C 180,E1 -18129.681,E2 -18129.681} C_VEL
LIN {X 0,Y 266.148,Z 758.837,A -85,B 0,C 180,E1 -18133.899,E2 -18133.899} C_VEL
LIN {X 0,Y 264.485,Z 750.532,A -85,B 0,C 180,E1 -18138.371,E2 -18138.371} C_VEL
LIN {X 0,Y 263.18,Z 743.7,A -85,B 0,C 180,E1 -18142.345,E2 -18142.345} C_VEL
LIN {X 0,Y 263.168,Z 743.705,A -85,B 0,C 180,E1 -18145.888,E2 -18145.888} C_VEL
LIN {X 0,Y 263.152,Z 743.706,A -85,B 0,C 180,E1 -18149.507,E2 -18149.507} C_VEL
LIN {X 0,Y 263.193,Z 743.695,A -85,B 0,C 180,E1 -18153.003,E2 -18153.003} C_VEL
LIN {X 0,Y 263.157,Z 743.704,A -85,B 0,C 180,E1 -18156.385,E2 -18156.385} C_VEL
LIN {X 0,Y 263.264,Z 743.69,A -85,B 0,C 180,E1 -18159.694,E2 -18159.694} C_VEL
LIN {X 0,Y 263.353,Z 743.68,A -85,B 0,C 180,E1 -18164.522,E2 -18164.522} C_VEL
LIN {X 0,Y 263.357,Z 743.676,A -85,B 0,C 180,E1 -18169.234,E2 -18169.234} C_VEL
LIN {X 0,Y 263.56,Z 743.655,A -85,B 0,C 180,E1 -18172.338,E2 -18172.338} C_VEL
LIN {X 0,Y 263.749,Z 743.631,A -85,B 0,C 180,E1 -18178.473,E2 -18178.473} C_VEL
LIN {X 0,Y 263.75,Z 743.628,A -85,B 0,C 180,E1 -18181.527,E2 -18181.527} C_VEL
LIN {X 0,Y 263.531,Z 743.654,A -85,B 0,C 180,E1 -18187.663,E2 -18187.663} C_VEL
LIN {X 0,Y 263.351,Z 743.681,A -85,B 0,C 180,E1 -18190.767,E2 -18190.767} C_VEL
LIN {X 0,Y 263.325,Z 743.681,A -85,B 0,C 180,E1 -18195.48,E2 -18195.48} C_VEL
LIN {X 0,Y 263.239,Z 743.692,A -85,B 0,C 180,E1 -18200.309,E2 -18200.309} C_VEL
LIN {X 0,Y 263.127,Z 743.708,A -85,B 0,C 180,E1 -18205.3,E2 -18205.3} C_VEL
LIN {X 0,Y 263.134,Z 743.705,A -85,B 0,C 180,E1 -18208.735,E2 -18208.735} C_VEL
LIN {X 0,Y 263.129,Z 743.705,A -85,B 0,C 180,E1 -18212.289,E2 -18212.289} C_VEL
LIN {X 0,Y 263.155,Z 743.705,A -85,B 0,C 180,E1 -18215.984,E2 -18215.984} C_VEL
LIN {X 0,Y 263.073,Z 743.716,A -85,B 0,C 180,E1 -18219.879,E2 -18219.879} C_VEL
LIN {X 0,Y 263.077,Z 743.716,A -85,B 0,C 180,E1 -18223.994,E2 -18223.994} C_VEL
LIN {X 0,Y 263.075,Z 743.714,A -85,B 0,C 180,E1 -18228.419,E2 -18228.419} C_VEL
LIN {X 0,Y 263.104,Z 743.712,A -85,B 0,C 180,E1 -18232.094,E2 -18232.094} C_VEL
LIN {X 0,Y 263.153,Z 743.705,A -85,B 0,C 180,E1 -18235.886,E2 -18235.886} C_VEL
LIN {X 0,Y 263.11,Z 743.706,A -85,B 0,C 180,E1 -18239.502,E2 -18239.502} C_VEL
LIN {X 0,Y 263.114,Z 743.708,A -85,B 0,C 180,E1 -18242.994,E2 -18242.994} C_VEL
LIN {X 0,Y 263.118,Z 743.711,A -85,B 0,C 180,E1 -18246.381,E2 -18246.381} C_VEL
LIN {X 0,Y 263.238,Z 743.691,A -85,B 0,C 180,E1 -18249.691,E2 -18249.691} C_VEL
LIN {X 0,Y 263.313,Z 743.686,A -85,B 0,C 180,E1 -18254.52,E2 -18254.52} C_VEL
LIN {X 0,Y 263.348,Z 743.68,A -85,B 0,C 180,E1 -18259.233,E2 -18259.233} C_VEL
LIN {X 0,Y 263.528,Z 743.657,A -85,B 0,C 180,E1 -18262.337,E2 -18262.337} C_VEL
LIN {X 0,Y 263.739,Z 743.63,A -85,B 0,C 180,E1 -18268.473,E2 -18268.473} C_VEL
LIN {X 0,Y 263.736,Z 743.632,A -85,B 0,C 180,E1 -18271.527,E2 -18271.527} C_VEL
LIN {X 0,Y 263.529,Z 743.658,A -85,B 0,C 180,E1 -18277.663,E2 -18277.663} C_VEL
LIN {X 0,Y 263.353,Z 743.678,A -85,B 0,C 180,E1 -18280.767,E2 -18280.767} C_VEL
LIN {X 0,Y 263.354,Z 743.681,A -85,B 0,C 180,E1 -18285.478,E2 -18285.478} C_VEL
LIN {X 0,Y 263.265,Z 743.688,A -85,B 0,C 180,E1 -18290.307,E2 -18290.307} C_VEL
LIN {X 0,Y 263.171,Z 743.701,A -85,B 0,C 180,E1 -18295.295,E2 -18295.295} C_VEL
LIN {X 0,Y 263.137,Z 743.705,A -85,B 0,C 180,E1 -18298.735,E2 -18298.735} C_VEL
LIN {X 0,Y 263.131,Z 743.709,A -85,B 0,C 180,E1 -18302.289,E2 -18302.289} C_VEL
LIN {X 0,Y 263.196,Z 743.699,A -85,B 0,C 180,E1 -18306.766,E2 -18306.766} C_VEL
LIN {X 0,Y 263.221,Z 743.719,A -85,B 0,C 180,E1 -18308.738,E2 -18308.738} C_VEL
LIN {X 0,Y 267.16,Z 756.999,A -85,B 0,C 180,E1 -18310.28,E2 -18310.28} C_VEL
LIN {X 0,Y 270.113,Z 767.979,A -85,B 0,C 180,E1 -18311.816,E2 -18311.816} C_VEL
LIN {X 0,Y 270.556,Z 770.116,A -85,B 0,C 180,E1 -18312.142,E2 -18312.142} C_VEL
LIN {X 0,Y 269.45,Z 780.537,A -85,B 0,C 180,E1 -18313.685,E2 -18313.685} C_VEL
LIN {X 0,Y 268.206,Z 790.527,A -85,B 0,C 180,E1 -18315.496,E2 -18315.496} C_VEL
LIN {X 0,Y 267.031,Z 799.441,A -85,B 0,C 180,E1 -18317.471,E2 -18317.471} C_VEL
LIN {X 0,Y 266.022,Z 807.146,A -85,B 0,C 180,E1 -18319.544,E2 -18319.544} C_VEL
LIN {X 0,Y 265.092,Z 814.404,A -85,B 0,C 180,E1 -18321.946,E2 -18321.946} C_VEL
LIN {X 0,Y 264.454,Z 819.861,A -85,B 0,C 180,E1 -18324.221,E2 -18324.221} C_VEL
LIN {X 0,Y 263.972,Z 824.853,A -85,B 0,C 180,E1 -18326.921,E2 -18326.921} C_VEL
LIN {X 0,Y 263.774,Z 828.406,A -85,B 0,C 180,E1 -18329.586,E2 -18329.586} C_VEL
LIN {X 0,Y 263.815,Z 830.16,A -85,B 0,C 180,E1 -18331.537,E2 -18331.537} C_VEL
LIN {X 0,Y 263.991,Z 831.099,A -85,B 0,C 180,E1 -18333.091,E2 -18333.091} C_VEL
LIN {X 0,Y 264.323,Z 831.659,A -85,B 0,C 180,E1 -18334.822,E2 -18334.822} C_VEL
LIN {X 0,Y 264.784,Z 831.687,A -85,B 0,C 180,E1 -18336.538,E2 -18336.538} C_VEL
LIN {X 0,Y 265.401,Z 831.251,A -85,B 0,C 180,E1 -18338.239,E2 -18338.239} C_VEL
LIN {X 0,Y 266.144,Z 830.268,A -85,B 0,C 180,E1 -18339.922,E2 -18339.922} C_VEL
LIN {X 0,Y 266.986,Z 828.842,A -85,B 0,C 180,E1 -18341.586,E2 -18341.586} C_VEL
LIN {X 0,Y 268.522,Z 825.728,A -85,B 0,C 180,E1 -18344.049,E2 -18344.049} C_VEL
LIN {X 0,Y 270.348,Z 821.406,A -85,B 0,C 180,E1 -18346.469,E2 -18346.469} C_VEL
LIN {X 0,Y 272.655,Z 815.442,A -85,B 0,C 180,E1 -18348.953,E2 -18348.953} C_VEL
LIN {X 0,Y 275.092,Z 808.518,A -85,B 0,C 180,E1 -18351.182,E2 -18351.182} C_VEL
LIN {X 0,Y 277.342,Z 801.128,A -85,B 0,C 180,E1 -18353.086,E2 -18353.086} C_VEL
LIN {X 0,Y 279.795,Z 792.181,A -85,B 0,C 180,E1 -18354.956,E2 -18354.956} C_VEL
LIN {X 0,Y 281.266,Z 785.972,A -85,B 0,C 180,E1 -18356.06,E2 -18356.06} C_VEL
LIN {X 0,Y 279.94,Z 779.326,A -85,B 0,C 180,E1 -18357.577,E2 -18357.577} C_VEL
LIN {X 0,Y 276.615,Z 768.69,A -85,B 0,C 180,E1 -18360,E2 -18360} C_VEL
LIN {X 0,Y 273.177,Z 760.432,A -85,B 0,C 180,E1 -18361.88,E2 -18361.88} C_VEL
LIN {X 0,Y 268.757,Z 752.727,A -85,B 0,C 180,E1 -18363.823,E2 -18363.823} C_VEL
LIN {X 0,Y 266.794,Z 749.789,A -85,B 0,C 180,E1 -18364.627,E2 -18364.627} C_VEL
LIN {X 0,Y 266.05,Z 748.365,A -85,B 0,C 180,E1 -18364.972,E2 -18364.972} C_VEL
LIN {X 0,Y 264.2,Z 746.054,A -85,B 0,C 180,E1 -18365.677,E2 -18365.677} C_VEL
LIN {X 0,Y 263.52,Z 743.651,A -85,B 0,C 180,E1 -18366.124,E2 -18366.124} C_VEL
LIN {X 0,Y 263.492,Z 743.654,A -85,B 0,C 180,E1 -18369.287,E2 -18369.287} C_VEL
LIN {X 0,Y 263.312,Z 743.684,A -85,B 0,C 180,E1 -18373.899,E2 -18373.899} C_VEL
LIN {X 0,Y 263.274,Z 743.688,A -85,B 0,C 180,E1 -18377.076,E2 -18377.076} C_VEL
LIN {X 0,Y 263.18,Z 743.694,A -85,B 0,C 180,E1 -18381.314,E2 -18381.314} C_VEL
LIN {X 0,Y 263.163,Z 743.764,A -85,B 0,C 180,E1 -18381.677,E2 -18381.677} C_VEL
LIN {X 0,Y 262.607,Z 744.516,A -85,B 0,C 180,E1 -18382.948,E2 -18382.948} C_VEL
LIN {X 0,Y 260.126,Z 746.44,A -85,B 0,C 180,E1 -18385.011,E2 -18385.011} C_VEL
LIN {X 0,Y 258.064,Z 748.143,A -85,B 0,C 180,E1 -18386.681,E2 -18386.681} C_VEL
LIN {X 0,Y 257.269,Z 749.261,A -85,B 0,C 180,E1 -18387.974,E2 -18387.974} C_VEL
LIN {X 0,Y 257.252,Z 749.568,A -85,B 0,C 180,E1 -18388.412,E2 -18388.412} C_VEL
LIN {X 0,Y 257.924,Z 752.464,A -85,B 0,C 180,E1 -18392.36,E2 -18392.36} C_VEL
LIN {X 0,Y 258.761,Z 756.446,A -85,B 0,C 180,E1 -18396.693,E2 -18396.693} C_VEL
LIN {X 0,Y 259.713,Z 760.666,A -85,B 0,C 180,E1 -18400.501,E2 -18400.501} C_VEL
LIN {X 0,Y 260.719,Z 765.825,A -85,B 0,C 180,E1 -18404.496,E2 -18404.496} C_VEL
LIN {X 0,Y 261.777,Z 772.139,A -85,B 0,C 180,E1 -18408.74,E2 -18408.74} C_VEL
LIN {X 0,Y 262.069,Z 774.083,A -85,B 0,C 180,E1 -18409.938,E2 -18409.938} C_VEL
LIN {X 0,Y 261.956,Z 776.07,A -85,B 0,C 180,E1 -18411.081,E2 -18411.081} C_VEL
LIN {X 0,Y 260.09,Z 783.204,A -85,B 0,C 180,E1 -18414.775,E2 -18414.775} C_VEL
LIN {X 0,Y 260.97,Z 787.369,A -85,B 0,C 180,E1 -18415.315,E2 -18415.315} C_VEL
LIN {X 0,Y 261.776,Z 790.111,A -85,B 0,C 180,E1 -18415.713,E2 -18415.713} C_VEL
LIN {X 0,Y 264.006,Z 799.145,A -85,B 0,C 180,E1 -18416.995,E2 -18416.995} C_VEL
LIN {X 0,Y 266.379,Z 814.07,A -85,B 0,C 180,E1 -18419.041,E2 -18419.041} C_VEL
LIN {X 0,Y 267.167,Z 826.393,A -85,B 0,C 180,E1 -18420.767,E2 -18420.767} C_VEL
LIN {X 0,Y 266.833,Z 839.771,A -85,B 0,C 180,E1 -18422.765,E2 -18422.765} C_VEL
LIN {X 0,Y 265.475,Z 850.879,A -85,B 0,C 180,E1 -18424.603,E2 -18424.603} C_VEL
LIN {X 0,Y 263.374,Z 862.25,A -85,B 0,C 180,E1 -18426.821,E2 -18426.821} C_VEL
LIN {X 0,Y 262.092,Z 869.006,A -85,B 0,C 180,E1 -18428.364,E2 -18428.364} C_VEL
LIN {X 0,Y 259.493,Z 877.622,A -85,B 0,C 180,E1 -18430.623,E2 -18430.623} C_VEL
LIN {X 0,Y 257.345,Z 885.182,A -85,B 0,C 180,E1 -18433.084,E2 -18433.084} C_VEL
LIN {X 0,Y 256.07,Z 891.572,A -85,B 0,C 180,E1 -18435.699,E2 -18435.699} C_VEL
LIN {X 0,Y 255.24,Z 896.215,A -85,B 0,C 180,E1 -18438.082,E2 -18438.082} C_VEL
LIN {X 0,Y 254.926,Z 899.848,A -85,B 0,C 180,E1 -18440.479,E2 -18440.479} C_VEL
LIN {X 0,Y 254.994,Z 902.508,A -85,B 0,C 180,E1 -18442.845,E2 -18442.845} C_VEL
LIN {X 0,Y 255.312,Z 904.313,A -85,B 0,C 180,E1 -18445.263,E2 -18445.263} C_VEL
LIN {X 0,Y 255.561,Z 904.983,A -85,B 0,C 180,E1 -18446.847,E2 -18446.847} C_VEL
LIN {X 0,Y 255.802,Z 905.233,A -85,B 0,C 180,E1 -18448.425,E2 -18448.425} C_VEL
LIN {X 0,Y 256.176,Z 905.039,A -85,B 0,C 180,E1 -18450,E2 -18450} C_VEL
LIN {X 0,Y 255.968,Z 904.313,A -85,B 0,C 180,E1 -18451.573,E2 -18451.573} C_VEL
LIN {X 0,Y 255.776,Z 903.158,A -85,B 0,C 180,E1 -18453.15,E2 -18453.15} C_VEL
LIN {X 0,Y 255.594,Z 900.538,A -85,B 0,C 180,E1 -18455.522,E2 -18455.522} C_VEL
LIN {X 0,Y 255.365,Z 896.774,A -85,B 0,C 180,E1 -18457.909,E2 -18457.909} C_VEL
LIN {X 0,Y 255.383,Z 891.817,A -85,B 0,C 180,E1 -18460.304,E2 -18460.304} C_VEL
LIN {X 0,Y 255.82,Z 885.551,A -85,B 0,C 180,E1 -18462.696,E2 -18462.696} C_VEL
LIN {X 0,Y 256.659,Z 877.675,A -85,B 0,C 180,E1 -18465.078,E2 -18465.078} C_VEL
LIN {X 0,Y 258.012,Z 867.945,A -85,B 0,C 180,E1 -18467.435,E2 -18467.435} C_VEL
LIN {X 0,Y 259.232,Z 858.942,A -85,B 0,C 180,E1 -18469.191,E2 -18469.191} C_VEL
LIN {X 0,Y 259.198,Z 847.327,A -85,B 0,C 180,E1 -18471.055,E2 -18471.055} C_VEL
LIN {X 0,Y 258.914,Z 835.126,A -85,B 0,C 180,E1 -18472.646,E2 -18472.646} C_VEL
LIN {X 0,Y 258.217,Z 821.994,A -85,B 0,C 180,E1 -18473.993,E2 -18473.993} C_VEL
LIN {X 0,Y 257.285,Z 808.229,A -85,B 0,C 180,E1 -18475.074,E2 -18475.074} C_VEL
LIN {X 0,Y 256.408,Z 797.741,A -85,B 0,C 180,E1 -18475.707,E2 -18475.707} C_VEL
LIN {X 0,Y 257.812,Z 787.913,A -85,B 0,C 180,E1 -18480.286,E2 -18480.286} C_VEL
LIN {X 0,Y 259.905,Z 776.215,A -85,B 0,C 180,E1 -18485.785,E2 -18485.785} C_VEL
LIN {X 0,Y 260.933,Z 770.242,A -85,B 0,C 180,E1 -18488.639,E2 -18488.639} C_VEL
LIN {X 0,Y 260.324,Z 765.761,A -85,B 0,C 180,E1 -18490.894,E2 -18490.894} C_VEL
LIN {X 0,Y 258.724,Z 757.91,A -85,B 0,C 180,E1 -18495.068,E2 -18495.068} C_VEL
LIN {X 0,Y 257.022,Z 749.194,A -85,B 0,C 180,E1 -18499.963,E2 -18499.963} C_VEL
LIN {X 0,Y 256.144,Z 744.576,A -85,B 0,C 180,E1 -18502.721,E2 -18502.721} C_VEL
LIN {X 0,Y 256.077,Z 744.584,A -85,B 0,C 180,E1 -18506.709,E2 -18506.709} C_VEL
LIN {X 0,Y 256.14,Z 744.577,A -85,B 0,C 180,E1 -18511.405,E2 -18511.405} C_VEL
LIN {X 0,Y 256.144,Z 744.578,A -85,B 0,C 180,E1 -18515.697,E2 -18515.697} C_VEL
LIN {X 0,Y 256.164,Z 744.573,A -85,B 0,C 180,E1 -18519.105,E2 -18519.105} C_VEL
LIN {X 0,Y 256.302,Z 744.559,A -85,B 0,C 180,E1 -18524.085,E2 -18524.085} C_VEL
LIN {X 0,Y 256.297,Z 744.557,A -85,B 0,C 180,E1 -18527.328,E2 -18527.328} C_VEL
LIN {X 0,Y 256.517,Z 744.53,A -85,B 0,C 180,E1 -18532.126,E2 -18532.126} C_VEL
LIN {X 0,Y 256.489,Z 744.534,A -85,B 0,C 180,E1 -18536.859,E2 -18536.859} C_VEL
LIN {X 0,Y 256.752,Z 744.499,A -85,B 0,C 180,E1 -18540,E2 -18540} C_VEL
LIN {X 0,Y 256.493,Z 744.534,A -85,B 0,C 180,E1 -18543.142,E2 -18543.142} C_VEL
LIN {X 0,Y 256.472,Z 744.533,A -85,B 0,C 180,E1 -18547.875,E2 -18547.875} C_VEL
LIN {X 0,Y 256.292,Z 744.562,A -85,B 0,C 180,E1 -18551.067,E2 -18551.067} C_VEL
LIN {X 0,Y 256.26,Z 744.559,A -85,B 0,C 180,E1 -18555.918,E2 -18555.918} C_VEL
LIN {X 0,Y 256.146,Z 744.578,A -85,B 0,C 180,E1 -18560.897,E2 -18560.897} C_VEL
LIN {X 0,Y 256.086,Z 744.584,A -85,B 0,C 180,E1 -18565.089,E2 -18565.089} C_VEL
LIN {X 0,Y 256.091,Z 744.582,A -85,B 0,C 180,E1 -18568.575,E2 -18568.575} C_VEL
LIN {X 0,Y 256.075,Z 744.587,A -85,B 0,C 180,E1 -18571.702,E2 -18571.702} C_VEL
LIN {X 0,Y 256.079,Z 744.584,A -85,B 0,C 180,E1 -18575.194,E2 -18575.194} C_VEL
LIN {X 0,Y 256.043,Z 744.589,A -85,B 0,C 180,E1 -18579.148,E2 -18579.148} C_VEL
LIN {X 0,Y 256.022,Z 744.59,A -85,B 0,C 180,E1 -18583.336,E2 -18583.336} C_VEL
LIN {X 0,Y 256.032,Z 744.593,A -85,B 0,C 180,E1 -18587.829,E2 -18587.829} C_VEL
LIN {X 0,Y 256.043,Z 744.586,A -85,B 0,C 180,E1 -18590.853,E2 -18590.853} C_VEL
LIN {X 0,Y 256.079,Z 744.585,A -85,B 0,C 180,E1 -18594.807,E2 -18594.807} C_VEL
LIN {X 0,Y 256.079,Z 744.584,A -85,B 0,C 180,E1 -18598.571,E2 -18598.571} C_VEL
LIN {X 0,Y 256.079,Z 744.586,A -85,B 0,C 180,E1 -18602.189,E2 -18602.189} C_VEL
LIN {X 0,Y 256.087,Z 744.583,A -85,B 0,C 180,E1 -18605.691,E2 -18605.691} C_VEL
LIN {X 0,Y 256.146,Z 744.575,A -85,B 0,C 180,E1 -18609.103,E2 -18609.103} C_VEL
LIN {X 0,Y 256.247,Z 744.564,A -85,B 0,C 180,E1 -18614.082,E2 -18614.082} C_VEL
LIN {X 0,Y 256.289,Z 744.562,A -85,B 0,C 180,E1 -18618.933,E2 -18618.933} C_VEL
LIN {X 0,Y 256.47,Z 744.535,A -85,B 0,C 180,E1 -18622.125,E2 -18622.125} C_VEL
LIN {X 0,Y 256.452,Z 744.539,A -85,B 0,C 180,E1 -18626.858,E2 -18626.858} C_VEL
LIN {X 0,Y 256.701,Z 744.506,A -85,B 0,C 180,E1 -18628.431,E2 -18628.431} C_VEL
LIN {X 0,Y 256.699,Z 744.508,A -85,B 0,C 180,E1 -18631.569,E2 -18631.569} C_VEL
LIN {X 0,Y 256.458,Z 744.536,A -85,B 0,C 180,E1 -18636.293,E2 -18636.293} C_VEL
LIN {X 0,Y 256.43,Z 744.545,A -85,B 0,C 180,E1 -18639.465,E2 -18639.465} C_VEL
LIN {X 0,Y 256.258,Z 744.561,A -85,B 0,C 180,E1 -18644.29,E2 -18644.29} C_VEL
LIN {X 0,Y 256.213,Z 744.572,A -85,B 0,C 180,E1 -18647.562,E2 -18647.562} C_VEL
LIN {X 0,Y 256.155,Z 744.574,A -85,B 0,C 180,E1 -18651.117,E2 -18651.117} C_VEL
LIN {X 0,Y 256.136,Z 744.577,A -85,B 0,C 180,E1 -18655.112,E2 -18655.112} C_VEL
LIN {X 0,Y 256.058,Z 744.589,A -85,B 0,C 180,E1 -18659.607,E2 -18659.607} C_VEL
LIN {X 0,Y 256.069,Z 744.586,A -85,B 0,C 180,E1 -18663.293,E2 -18663.293} C_VEL
LIN {X 0,Y 256.14,Z 744.577,A -85,B 0,C 180,E1 -18667.278,E2 -18667.278} C_VEL
LIN {X 0,Y 256.146,Z 744.582,A -85,B 0,C 180,E1 -18668.284,E2 -18668.284} C_VEL
LIN {X 0,Y 259.785,Z 756.873,A -85,B 0,C 180,E1 -18669.748,E2 -18669.748} C_VEL
LIN {X 0,Y 262.546,Z 766.742,A -85,B 0,C 180,E1 -18671.139,E2 -18671.139} C_VEL
LIN {X 0,Y 263.606,Z 770.982,A -85,B 0,C 180,E1 -18671.8,E2 -18671.8} C_VEL
LIN {X 0,Y 262.532,Z 781.72,A -85,B 0,C 180,E1 -18673.436,E2 -18673.436} C_VEL
LIN {X 0,Y 261.199,Z 791.915,A -85,B 0,C 180,E1 -18675.343,E2 -18675.343} C_VEL
LIN {X 0,Y 259.932,Z 801.196,A -85,B 0,C 180,E1 -18677.472,E2 -18677.472} C_VEL
LIN {X 0,Y 258.778,Z 809.75,A -85,B 0,C 180,E1 -18679.9,E2 -18679.9} C_VEL
LIN {X 0,Y 257.79,Z 817.408,A -85,B 0,C 180,E1 -18682.664,E2 -18682.664} C_VEL
LIN {X 0,Y 257.261,Z 822.558,A -85,B 0,C 180,E1 -18685.041,E2 -18685.041} C_VEL
LIN {X 0,Y 256.844,Z 827.402,A -85,B 0,C 180,E1 -18688.023,E2 -18688.023} C_VEL
LIN {X 0,Y 256.77,Z 830.823,A -85,B 0,C 180,E1 -18691.149,E2 -18691.149} C_VEL
LIN {X 0,Y 257.15,Z 832.496,A -85,B 0,C 180,E1 -18694.069,E2 -18694.069} C_VEL
LIN {X 0,Y 257.576,Z 832.858,A -85,B 0,C 180,E1 -18695.84,E2 -18695.84} C_VEL
LIN {X 0,Y 258.189,Z 832.664,A -85,B 0,C 180,E1 -18697.744,E2 -18697.744} C_VEL
LIN {X 0,Y 258.859,Z 832.043,A -85,B 0,C 180,E1 -18699.332,E2 -18699.332} C_VEL
LIN {X 0,Y 259.797,Z 830.775,A -85,B 0,C 180,E1 -18701.231,E2 -18701.231} C_VEL
LIN {X 0,Y 261.178,Z 828.312,A -85,B 0,C 180,E1 -18703.588,E2 -18703.588} C_VEL
LIN {X 0,Y 263.024,Z 824.492,A -85,B 0,C 180,E1 -18706.085,E2 -18706.085} C_VEL
LIN {X 0,Y 265.299,Z 819.292,A -85,B 0,C 180,E1 -18708.571,E2 -18708.571} C_VEL
LIN {X 0,Y 267.794,Z 812.872,A -85,B 0,C 180,E1 -18710.94,E2 -18710.94} C_VEL
LIN {X 0,Y 270.631,Z 804.582,A -85,B 0,C 180,E1 -18713.307,E2 -18713.307} C_VEL
LIN {X 0,Y 273.193,Z 796.216,A -85,B 0,C 180,E1 -18715.204,E2 -18715.204} C_VEL
LIN {X 0,Y 275.194,Z 788.431,A -85,B 0,C 180,E1 -18716.668,E2 -18716.668} C_VEL
LIN {X 0,Y 273.701,Z 780.873,A -85,B 0,C 180,E1 -18718.528,E2 -18718.528} C_VEL
LIN {X 0,Y 270.286,Z 769.78,A -85,B 0,C 180,E1 -18721.198,E2 -18721.198} C_VEL
LIN {X 0,Y 267.093,Z 762.638,A -85,B 0,C 180,E1 -18723.016,E2 -18723.016} C_VEL
LIN {X 0,Y 264.618,Z 758.171,A -85,B 0,C 180,E1 -18724.237,E2 -18724.237} C_VEL
LIN {X 0,Y 262.966,Z 755.704,A -85,B 0,C 180,E1 -18724.983,E2 -18724.983} C_VEL
LIN {X 0,Y 262.223,Z 754.095,A -85,B 0,C 180,E1 -18725.383,E2 -18725.383} C_VEL
LIN {X 0,Y 260.13,Z 751.092,A -85,B 0,C 180,E1 -18726.301,E2 -18726.301} C_VEL
LIN {X 0,Y 259.384,Z 749.404,A -85,B 0,C 180,E1 -18726.71,E2 -18726.71} C_VEL
LIN {X 0,Y 257.405,Z 747.177,A -85,B 0,C 180,E1 -18727.55,E2 -18727.55} C_VEL
LIN {X 0,Y 256.551,Z 744.852,A -85,B 0,C 180,E1 -18728.043,E2 -18728.043} C_VEL
LIN {X 0,Y 256.494,Z 744.529,A -85,B 0,C 180,E1 -18728.148,E2 -18728.148} C_VEL
LIN {X 0,Y 256.298,Z 744.552,A -85,B 0,C 180,E1 -18732.672,E2 -18732.672} C_VEL
LIN {X 0,Y 256.286,Z 744.569,A -85,B 0,C 180,E1 -18736.302,E2 -18736.302} C_VEL
LIN {X 0,Y 256.467,Z 745.983,A -85,B 0,C 180,E1 -18741.296,E2 -18741.296} C_VEL
LIN {X 0,Y 256.939,Z 748.077,A -85,B 0,C 180,E1 -18745.954,E2 -18745.954} C_VEL
LIN {X 0,Y 257.252,Z 749.568,A -85,B 0,C 180,E1 -18748.412,E2 -18748.412} C_VEL
LIN {X 0,Y 256.802,Z 750.666,A -85,B 0,C 180,E1 -18749.702,E2 -18749.702} C_VEL
LIN {X 0,Y 254.404,Z 753.175,A -85,B 0,C 180,E1 -18751.786,E2 -18751.786} C_VEL
LIN {X 0,Y 252.392,Z 755.359,A -85,B 0,C 180,E1 -18753.472,E2 -18753.472} C_VEL
LIN {X 0,Y 251.666,Z 756.857,A -85,B 0,C 180,E1 -18754.778,E2 -18754.778} C_VEL
LIN {X 0,Y 251.685,Z 757.285,A -85,B 0,C 180,E1 -18755.221,E2 -18755.221} C_VEL
LIN {X 0,Y 252.783,Z 761.913,A -85,B 0,C 180,E1 -18759.751,E2 -18759.751} C_VEL
LIN {X 0,Y 253.77,Z 767.089,A -85,B 0,C 180,E1 -18763.941,E2 -18763.941} C_VEL
LIN {X 0,Y 254.495,Z 771.527,A -85,B 0,C 180,E1 -18767.101,E2 -18767.101} C_VEL
LIN {X 0,Y 255.118,Z 775.416,A -85,B 0,C 180,E1 -18769.656,E2 -18769.656} C_VEL
LIN {X 0,Y 255.071,Z 777.127,A -85,B 0,C 180,E1 -18770.674,E2 -18770.674} C_VEL
LIN {X 0,Y 253.991,Z 781.517,A -85,B 0,C 180,E1 -18773.026,E2 -18773.026} C_VEL
LIN {X 0,Y 254.93,Z 785.77,A -85,B 0,C 180,E1 -18773.623,E2 -18773.623} C_VEL
LIN {X 0,Y 255.626,Z 788.003,A -85,B 0,C 180,E1 -18774,E2 -18774} C_VEL
LIN {X 0,Y 258.665,Z 801.632,A -85,B 0,C 180,E1 -18776.088,E2 -18776.088} C_VEL
LIN {X 0,Y 260.468,Z 814.638,A -85,B 0,C 180,E1 -18778.012,E2 -18778.012} C_VEL
LIN {X 0,Y 261.142,Z 828.071,A -85,B 0,C 180,E1 -18780.024,E2 -18780.024} C_VEL
LIN {X 0,Y 260.642,Z 839.505,A -85,B 0,C 180,E1 -18781.844,E2 -18781.844} C_VEL
LIN {X 0,Y 259.31,Z 849.911,A -85,B 0,C 180,E1 -18783.659,E2 -18783.659} C_VEL
LIN {X 0,Y 257.199,Z 860.668,A -85,B 0,C 180,E1 -18785.803,E2 -18785.803} C_VEL
LIN {X 0,Y 255.463,Z 868.949,A -85,B 0,C 180,E1 -18787.773,E2 -18787.773} C_VEL
LIN {X 0,Y 252.766,Z 877.335,A -85,B 0,C 180,E1 -18790.086,E2 -18790.086} C_VEL
LIN {X 0,Y 250.334,Z 885.306,A -85,B 0,C 180,E1 -18792.833,E2 -18792.833} C_VEL
LIN {X 0,Y 249.111,Z 890.95,A -85,B 0,C 180,E1 -18795.291,E2 -18795.291} C_VEL
LIN {X 0,Y 248.05,Z 896.739,A -85,B 0,C 180,E1 -18798.56,E2 -18798.56} C_VEL
LIN {X 0,Y 247.862,Z 899.012,A -85,B 0,C 180,E1 -18800.205,E2 -18800.205} C_VEL
LIN {X 0,Y 247.98,Z 902.266,A -85,B 0,C 180,E1 -18803.491,E2 -18803.491} C_VEL
LIN {X 0,Y 248.242,Z 903.306,A -85,B 0,C 180,E1 -18805.128,E2 -18805.128} C_VEL
LIN {X 0,Y 248.501,Z 903.935,A -85,B 0,C 180,E1 -18806.757,E2 -18806.757} C_VEL
LIN {X 0,Y 248.772,Z 904.112,A -85,B 0,C 180,E1 -18808.381,E2 -18808.381} C_VEL
LIN {X 0,Y 249.173,Z 903.877,A -85,B 0,C 180,E1 -18810,E2 -18810} C_VEL
LIN {X 0,Y 248.964,Z 903.116,A -85,B 0,C 180,E1 -18811.617,E2 -18811.617} C_VEL
LIN {X 0,Y 248.743,Z 901.914,A -85,B 0,C 180,E1 -18813.239,E2 -18813.239} C_VEL
LIN {X 0,Y 248.57,Z 899.204,A -85,B 0,C 180,E1 -18815.679,E2 -18815.679} C_VEL
LIN {X 0,Y 248.335,Z 895.337,A -85,B 0,C 180,E1 -18818.135,E2 -18818.135} C_VEL
LIN {X 0,Y 248.43,Z 889.265,A -85,B 0,C 180,E1 -18821.008,E2 -18821.008} C_VEL
LIN {X 0,Y 248.976,Z 882.602,A -85,B 0,C 180,E1 -18823.466,E2 -18823.466} C_VEL
LIN {X 0,Y 249.988,Z 874.338,A -85,B 0,C 180,E1 -18825.909,E2 -18825.909} C_VEL
LIN {X 0,Y 251.196,Z 865.677,A -85,B 0,C 180,E1 -18827.962,E2 -18827.962} C_VEL
LIN {X 0,Y 252.131,Z 858.945,A -85,B 0,C 180,E1 -18829.309,E2 -18829.309} C_VEL
LIN {X 0,Y 252.136,Z 847.488,A -85,B 0,C 180,E1 -18831.245,E2 -18831.245} C_VEL
LIN {X 0,Y 251.851,Z 834.636,A -85,B 0,C 180,E1 -18832.996,E2 -18832.996} C_VEL
LIN {X 0,Y 251.258,Z 821.87,A -85,B 0,C 180,E1 -18834.367,E2 -18834.367} C_VEL
LIN {X 0,Y 250.352,Z 807.937,A -85,B 0,C 180,E1 -18835.508,E2 -18835.508} C_VEL
LIN {X 0,Y 249.445,Z 796.786,A -85,B 0,C 180,E1 -18836.199,E2 -18836.199} C_VEL
LIN {X 0,Y 250.701,Z 788.273,A -85,B 0,C 180,E1 -18840.305,E2 -18840.305} C_VEL
LIN {X 0,Y 253.033,Z 775.809,A -85,B 0,C 180,E1 -18846.344,E2 -18846.344} C_VEL
LIN {X 0,Y 253.841,Z 771.733,A -85,B 0,C 180,E1 -18848.341,E2 -18848.341} C_VEL
LIN {X 0,Y 253.44,Z 767.52,A -85,B 0,C 180,E1 -18850.512,E2 -18850.512} C_VEL
LIN {X 0,Y 251.778,Z 759.345,A -85,B 0,C 180,E1 -18854.944,E2 -18854.944} C_VEL
LIN {X 0,Y 250.128,Z 750.997,A -85,B 0,C 180,E1 -18859.741,E2 -18859.741} C_VEL
LIN {X 0,Y 249.1,Z 745.454,A -85,B 0,C 180,E1 -18863.162,E2 -18863.162} C_VEL
LIN {X 0,Y 249.04,Z 745.466,A -85,B 0,C 180,E1 -18867.845,E2 -18867.845} C_VEL
LIN {X 0,Y 249.098,Z 745.454,A -85,B 0,C 180,E1 -18871.339,E2 -18871.339} C_VEL
LIN {X 0,Y 249.136,Z 745.448,A -85,B 0,C 180,E1 -18874.967,E2 -18874.967} C_VEL
LIN {X 0,Y 249.111,Z 745.454,A -85,B 0,C 180,E1 -18880.212,E2 -18880.212} C_VEL
LIN {X 0,Y 249.243,Z 745.435,A -85,B 0,C 180,E1 -18883.622,E2 -18883.622} C_VEL
LIN {X 0,Y 249.246,Z 745.436,A -85,B 0,C 180,E1 -18888.616,E2 -18888.616} C_VEL
LIN {X 0,Y 249.456,Z 745.408,A -85,B 0,C 180,E1 -18891.902,E2 -18891.902} C_VEL
LIN {X 0,Y 249.286,Z 745.431,A -85,B 0,C 180,E1 -18895.148,E2 -18895.148} C_VEL
LIN {X 0,Y 249.673,Z 745.384,A -85,B 0,C 180,E1 -18898.387,E2 -18898.387} C_VEL
LIN {X 0,Y 249.674,Z 745.381,A -85,B 0,C 180,E1 -18901.613,E2 -18901.613} C_VEL
LIN {X 0,Y 249.427,Z 745.413,A -85,B 0,C 180,E1 -18906.563,E2 -18906.563} C_VEL
LIN {X 0,Y 249.344,Z 745.423,A -85,B 0,C 180,E1 -18909.737,E2 -18909.737} C_VEL
LIN {X 0,Y 249.184,Z 745.444,A -85,B 0,C 180,E1 -18914.705,E2 -18914.705} C_VEL
LIN {X 0,Y 249.113,Z 745.451,A -85,B 0,C 180,E1 -18918.08,E2 -18918.08} C_VEL
LIN {X 0,Y 249.079,Z 745.458,A -85,B 0,C 180,E1 -18921.519,E2 -18921.519} C_VEL
LIN {X 0,Y 249.049,Z 745.462,A -85,B 0,C 180,E1 -18925.442,E2 -18925.442} C_VEL
LIN {X 0,Y 249.038,Z 745.462,A -85,B 0,C 180,E1 -18928.974,E2 -18928.974} C_VEL
LIN {X 0,Y 249.029,Z 745.461,A -85,B 0,C 180,E1 -18932.426,E2 -18932.426} C_VEL
LIN {X 0,Y 249.011,Z 745.465,A -85,B 0,C 180,E1 -18936.349,E2 -18936.349} C_VEL
LIN {X 0,Y 248.973,Z 745.469,A -85,B 0,C 180,E1 -18940.485,E2 -18940.485} C_VEL
LIN {X 0,Y 248.963,Z 745.47,A -85,B 0,C 180,E1 -18944.889,E2 -18944.889} C_VEL
LIN {X 0,Y 248.978,Z 745.469,A -85,B 0,C 180,E1 -18947.355,E2 -18947.355} C_VEL
LIN {X 0,Y 249.022,Z 745.466,A -85,B 0,C 180,E1 -18952.207,E2 -18952.207} C_VEL
LIN {X 0,Y 249.044,Z 745.461,A -85,B 0,C 180,E1 -18955.639,E2 -18955.639} C_VEL
LIN {X 0,Y 248.995,Z 745.464,A -85,B 0,C 180,E1 -18959.465,E2 -18959.465} C_VEL
LIN {X 0,Y 249.015,Z 745.464,A -85,B 0,C 180,E1 -18963.155,E2 -18963.155} C_VEL
LIN {X 0,Y 249.01,Z 745.466,A -85,B 0,C 180,E1 -18966.726,E2 -18966.726} C_VEL
LIN {X 0,Y 249.084,Z 745.456,A -85,B 0,C 180,E1 -18970.209,E2 -18970.209} C_VEL
LIN {X 0,Y 249.198,Z 745.441,A -85,B 0,C 180,E1 -18973.619,E2 -18973.619} C_VEL
LIN {X 0,Y 249.233,Z 745.438,A -85,B 0,C 180,E1 -18978.616,E2 -18978.616} C_VEL
LIN {X 0,Y 249.42,Z 745.413,A -85,B 0,C 180,E1 -18981.901,E2 -18981.901} C_VEL
LIN {X 0,Y 249.263,Z 745.434,A -85,B 0,C 180,E1 -18985.148,E2 -18985.148} C_VEL
LIN {X 0,Y 249.661,Z 745.383,A -85,B 0,C 180,E1 -18988.387,E2 -18988.387} C_VEL
LIN {X 0,Y 249.66,Z 745.385,A -85,B 0,C 180,E1 -18991.613,E2 -18991.613} C_VEL
LIN {X 0,Y 249.429,Z 745.412,A -85,B 0,C 180,E1 -18996.471,E2 -18996.471} C_VEL
LIN {X 0,Y 249.345,Z 745.425,A -85,B 0,C 180,E1 -18999.737,E2 -18999.737} C_VEL
LIN {X 0,Y 249.209,Z 745.439,A -85,B 0,C 180,E1 -19004.703,E2 -19004.703} C_VEL
LIN {X 0,Y 249.141,Z 745.45,A -85,B 0,C 180,E1 -19008.077,E2 -19008.077} C_VEL
LIN {X 0,Y 249.086,Z 745.457,A -85,B 0,C 180,E1 -19011.518,E2 -19011.518} C_VEL
LIN {X 0,Y 249.088,Z 745.456,A -85,B 0,C 180,E1 -19015.46,E2 -19015.46} C_VEL
LIN {X 0,Y 249.04,Z 745.461,A -85,B 0,C 180,E1 -19018.974,E2 -19018.974} C_VEL
LIN {X 0,Y 249.03,Z 745.465,A -85,B 0,C 180,E1 -19022.426,E2 -19022.426} C_VEL
LIN {X 0,Y 249.062,Z 745.462,A -85,B 0,C 180,E1 -19026.34,E2 -19026.34} C_VEL
LIN {X 0,Y 249.131,Z 745.657,A -85,B 0,C 180,E1 -19027.859,E2 -19027.859} C_VEL
LIN {X 0,Y 252.997,Z 758.665,A -85,B 0,C 180,E1 -19029.453,E2 -19029.453} C_VEL
LIN {X 0,Y 255.881,Z 769.072,A -85,B 0,C 180,E1 -19030.977,E2 -19030.977} C_VEL
LIN {X 0,Y 256.53,Z 771.612,A -85,B 0,C 180,E1 -19031.395,E2 -19031.395} C_VEL
LIN {X 0,Y 256.387,Z 775.29,A -85,B 0,C 180,E1 -19031.944,E2 -19031.944} C_VEL
LIN {X 0,Y 255.113,Z 786.547,A -85,B 0,C 180,E1 -19033.831,E2 -19033.831} C_VEL
LIN {X 0,Y 253.86,Z 795.706,A -85,B 0,C 180,E1 -19035.706,E2 -19035.706} C_VEL
LIN {X 0,Y 252.534,Z 805.15,A -85,B 0,C 180,E1 -19038.093,E2 -19038.093} C_VEL
LIN {X 0,Y 251.494,Z 812.758,A -85,B 0,C 180,E1 -19040.465,E2 -19040.465} C_VEL
LIN {X 0,Y 250.63,Z 819.134,A -85,B 0,C 180,E1 -19042.923,E2 -19042.923} C_VEL
LIN {X 0,Y 250.098,Z 824.893,A -85,B 0,C 180,E1 -19045.804,E2 -19045.804} C_VEL
LIN {X 0,Y 249.744,Z 829.111,A -85,B 0,C 180,E1 -19048.627,E2 -19048.627} C_VEL
LIN {X 0,Y 249.749,Z 831.972,A -85,B 0,C 180,E1 -19051.42,E2 -19051.42} C_VEL
LIN {X 0,Y 250.126,Z 833.519,A -85,B 0,C 180,E1 -19054.045,E2 -19054.045} C_VEL
LIN {X 0,Y 250.881,Z 833.989,A -85,B 0,C 180,E1 -19056.909,E2 -19056.909} C_VEL
LIN {X 0,Y 251.572,Z 833.654,A -85,B 0,C 180,E1 -19058.705,E2 -19058.705} C_VEL
LIN {X 0,Y 252.681,Z 832.463,A -85,B 0,C 180,E1 -19061.027,E2 -19061.027} C_VEL
LIN {X 0,Y 254.436,Z 829.725,A -85,B 0,C 180,E1 -19063.965,E2 -19063.965} C_VEL
LIN {X 0,Y 256.397,Z 826.005,A -85,B 0,C 180,E1 -19066.527,E2 -19066.527} C_VEL
LIN {X 0,Y 258.765,Z 821.02,A -85,B 0,C 180,E1 -19069.04,E2 -19069.04} C_VEL
LIN {X 0,Y 261.423,Z 814.656,A -85,B 0,C 180,E1 -19071.498,E2 -19071.498} C_VEL
LIN {X 0,Y 263.869,Z 808.097,A -85,B 0,C 180,E1 -19073.5,E2 -19073.5} C_VEL
LIN {X 0,Y 266.605,Z 800.103,A -85,B 0,C 180,E1 -19075.464,E2 -19075.464} C_VEL
LIN {X 0,Y 269.191,Z 790.887,A -85,B 0,C 180,E1 -19077.331,E2 -19077.331} C_VEL
LIN {X 0,Y 267.708,Z 783.32,A -85,B 0,C 180,E1 -19079.323,E2 -19079.323} C_VEL
LIN {X 0,Y 265.369,Z 774.771,A -85,B 0,C 180,E1 -19081.517,E2 -19081.517} C_VEL
LIN {X 0,Y 262.541,Z 767.838,A -85,B 0,C 180,E1 -19083.393,E2 -19083.393} C_VEL
LIN {X 0,Y 260.372,Z 763.547,A -85,B 0,C 180,E1 -19084.645,E2 -19084.645} C_VEL
LIN {X 0,Y 256.488,Z 757.062,A -85,B 0,C 180,E1 -19086.688,E2 -19086.688} C_VEL
LIN {X 0,Y 255.823,Z 755.485,A -85,B 0,C 180,E1 -19087.102,E2 -19087.102} C_VEL
LIN {X 0,Y 253.402,Z 752.016,A -85,B 0,C 180,E1 -19088.317,E2 -19088.317} C_VEL
LIN {X 0,Y 252.589,Z 750.494,A -85,B 0,C 180,E1 -19088.755,E2 -19088.755} C_VEL
LIN {X 0,Y 250.257,Z 748.132,A -85,B 0,C 180,E1 -19089.886,E2 -19089.886} C_VEL
LIN {X 0,Y 249.473,Z 746.332,A -85,B 0,C 180,E1 -19090.408,E2 -19090.408} C_VEL
LIN {X 0,Y 249.478,Z 746.677,A -85,B 0,C 180,E1 -19094.687,E2 -19094.687} C_VEL
LIN {X 0,Y 249.567,Z 747.329,A -85,B 0,C 180,E1 -19098.045,E2 -19098.045} C_VEL
LIN {X 0,Y 249.79,Z 748.543,A -85,B 0,C 180,E1 -19101.8,E2 -19101.8} C_VEL
LIN {X 0,Y 250.259,Z 750.478,A -85,B 0,C 180,E1 -19106.018,E2 -19106.018} C_VEL
LIN {X 0,Y 250.825,Z 753.195,A -85,B 0,C 180,E1 -19110.288,E2 -19110.288} C_VEL
LIN {X 0,Y 251.468,Z 756.134,A -85,B 0,C 180,E1 -19113.984,E2 -19113.984} C_VEL
LIN {X 0,Y 251.685,Z 757.285,A -85,B 0,C 180,E1 -19115.221,E2 -19115.221} C_VEL
LIN {X 0,Y 251.34,Z 758.745,A -85,B 0,C 180,E1 -19116.522,E2 -19116.522} C_VEL
LIN {X 0,Y 249.077,Z 761.8,A -85,B 0,C 180,E1 -19118.621,E2 -19118.621} C_VEL
LIN {X 0,Y 247.15,Z 764.408,A -85,B 0,C 180,E1 -19120.317,E2 -19120.317} C_VEL
LIN {X 0,Y 246.485,Z 766.231,A -85,B 0,C 180,E1 -19121.63,E2 -19121.63} C_VEL
LIN {X 0,Y 246.524,Z 766.781,A -85,B 0,C 180,E1 -19122.075,E2 -19122.075} C_VEL
LIN {X 0,Y 247.466,Z 772.083,A -85,B 0,C 180,E1 -19126.166,E2 -19126.166} C_VEL
LIN {X 0,Y 248.169,Z 776.741,A -85,B 0,C 180,E1 -19129.356,E2 -19129.356} C_VEL
LIN {X 0,Y 247.952,Z 779.484,A -85,B 0,C 180,E1 -19130.992,E2 -19130.992} C_VEL
LIN {X 0,Y 248.951,Z 783.92,A -85,B 0,C 180,E1 -19131.712,E2 -19131.712} C_VEL
LIN {X 0,Y 249.811,Z 786.598,A -85,B 0,C 180,E1 -19132.239,E2 -19132.239} C_VEL
LIN {X 0,Y 252.09,Z 796.807,A -85,B 0,C 180,E1 -19133.949,E2 -19133.949} C_VEL
LIN {X 0,Y 254.157,Z 809.757,A -85,B 0,C 180,E1 -19136.054,E2 -19136.054} C_VEL
LIN {X 0,Y 255.086,Z 821.739,A -85,B 0,C 180,E1 -19137.953,E2 -19137.953} C_VEL
LIN {X 0,Y 254.958,Z 834.399,A -85,B 0,C 180,E1 -19140.047,E2 -19140.047} C_VEL
LIN {X 0,Y 253.933,Z 845.123,A -85,B 0,C 180,E1 -19141.933,E2 -19141.933} C_VEL
LIN {X 0,Y 251.942,Z 855.435,A -85,B 0,C 180,E1 -19143.937,E2 -19143.937} C_VEL
LIN {X 0,Y 249.56,Z 865.884,A -85,B 0,C 180,E1 -19146.34,E2 -19146.34} C_VEL
LIN {X 0,Y 247.966,Z 871.833,A -85,B 0,C 180,E1 -19147.942,E2 -19147.942} C_VEL
LIN {X 0,Y 245.294,Z 879.516,A -85,B 0,C 180,E1 -19150.327,E2 -19150.327} C_VEL
LIN {X 0,Y 243.057,Z 886.829,A -85,B 0,C 180,E1 -19153.193,E2 -19153.193} C_VEL
LIN {X 0,Y 241.831,Z 891.927,A -85,B 0,C 180,E1 -19155.698,E2 -19155.698} C_VEL
LIN {X 0,Y 240.88,Z 897.109,A -85,B 0,C 180,E1 -19159.068,E2 -19159.068} C_VEL
LIN {X 0,Y 240.877,Z 900.909,A -85,B 0,C 180,E1 -19162.753,E2 -19162.753} C_VEL
LIN {X 0,Y 241.175,Z 902.305,A -85,B 0,C 180,E1 -19164.984,E2 -19164.984} C_VEL
LIN {X 0,Y 241.445,Z 902.855,A -85,B 0,C 180,E1 -19166.662,E2 -19166.662} C_VEL
LIN {X 0,Y 241.742,Z 902.972,A -85,B 0,C 180,E1 -19168.334,E2 -19168.334} C_VEL
LIN {X 0,Y 242.166,Z 902.695,A -85,B 0,C 180,E1 -19170,E2 -19170} C_VEL
LIN {X 0,Y 241.955,Z 901.889,A -85,B 0,C 180,E1 -19171.664,E2 -19171.664} C_VEL
LIN {X 0,Y 241.719,Z 900.602,A -85,B 0,C 180,E1 -19173.333,E2 -19173.333} C_VEL
LIN {X 0,Y 241.543,Z 897.805,A -85,B 0,C 180,E1 -19175.845,E2 -19175.845} C_VEL
LIN {X 0,Y 241.292,Z 893.819,A -85,B 0,C 180,E1 -19178.374,E2 -19178.374} C_VEL
LIN {X 0,Y 241.432,Z 887.611,A -85,B 0,C 180,E1 -19181.332,E2 -19181.332} C_VEL
LIN {X 0,Y 242.051,Z 880.83,A -85,B 0,C 180,E1 -19183.859,E2 -19183.859} C_VEL
LIN {X 0,Y 243.138,Z 872.353,A -85,B 0,C 180,E1 -19186.369,E2 -19186.369} C_VEL
LIN {X 0,Y 244.385,Z 863.692,A -85,B 0,C 180,E1 -19188.441,E2 -19188.441} C_VEL
LIN {X 0,Y 245.03,Z 858.65,A -85,B 0,C 180,E1 -19189.477,E2 -19189.477} C_VEL
LIN {X 0,Y 245.085,Z 847.537,A -85,B 0,C 180,E1 -19191.445,E2 -19191.445} C_VEL
LIN {X 0,Y 244.823,Z 834.636,A -85,B 0,C 180,E1 -19193.277,E2 -19193.277} C_VEL
LIN {X 0,Y 244.317,Z 822.533,A -85,B 0,C 180,E1 -19194.652,E2 -19194.652} C_VEL
LIN {X 0,Y 243.388,Z 808.244,A -85,B 0,C 180,E1 -19195.893,E2 -19195.893} C_VEL
LIN {X 0,Y 242.503,Z 795.894,A -85,B 0,C 180,E1 -19196.69,E2 -19196.69} C_VEL
LIN {X 0,Y 243.884,Z 786.739,A -85,B 0,C 180,E1 -19201.245,E2 -19201.245} C_VEL
LIN {X 0,Y 246.163,Z 775.401,A -85,B 0,C 180,E1 -19206.927,E2 -19206.927} C_VEL
LIN {X 0,Y 246.78,Z 771.736,A -85,B 0,C 180,E1 -19208.795,E2 -19208.795} C_VEL
LIN {X 0,Y 246.226,Z 767.541,A -85,B 0,C 180,E1 -19211.033,E2 -19211.033} C_VEL
LIN {X 0,Y 244.716,Z 760.153,A -85,B 0,C 180,E1 -19215.176,E2 -19215.176} C_VEL
LIN {X 0,Y 243.231,Z 752.724,A -85,B 0,C 180,E1 -19219.55,E2 -19219.55} C_VEL
LIN {X 0,Y 242.033,Z 746.334,A -85,B 0,C 180,E1 -19223.599,E2 -19223.599} C_VEL
LIN {X 0,Y 241.994,Z 746.341,A -85,B 0,C 180,E1 -19227.375,E2 -19227.375} C_VEL
LIN {X 0,Y 242.038,Z 746.333,A -85,B 0,C 180,E1 -19230.587,E2 -19230.587} C_VEL
LIN {X 0,Y 242.069,Z 746.331,A -85,B 0,C 180,E1 -19234.183,E2 -19234.183} C_VEL
LIN {X 0,Y 242.027,Z 746.337,A -85,B 0,C 180,E1 -19238.313,E2 -19238.313} C_VEL
LIN {X 0,Y 242.165,Z 746.316,A -85,B 0,C 180,E1 -19243.278,E2 -19243.278} C_VEL
LIN {X 0,Y 242.183,Z 746.319,A -85,B 0,C 180,E1 -19248.28,E2 -19248.28} C_VEL
LIN {X 0,Y 242.402,Z 746.286,A -85,B 0,C 180,E1 -19251.665,E2 -19251.665} C_VEL
LIN {X 0,Y 242.424,Z 746.285,A -85,B 0,C 180,E1 -19253.341,E2 -19253.341} C_VEL
LIN {X 0,Y 242.633,Z 746.26,A -85,B 0,C 180,E1 -19258.34,E2 -19258.34} C_VEL
LIN {X 0,Y 242.635,Z 746.258,A -85,B 0,C 180,E1 -19261.66,E2 -19261.66} C_VEL
LIN {X 0,Y 242.403,Z 746.29,A -85,B 0,C 180,E1 -19266.66,E2 -19266.66} C_VEL
LIN {X 0,Y 242.267,Z 746.304,A -85,B 0,C 180,E1 -19270.024,E2 -19270.024} C_VEL
LIN {X 0,Y 242.141,Z 746.322,A -85,B 0,C 180,E1 -19275.143,E2 -19275.143} C_VEL
LIN {X 0,Y 242.051,Z 746.331,A -85,B 0,C 180,E1 -19278.626,E2 -19278.626} C_VEL
LIN {X 0,Y 241.989,Z 746.339,A -85,B 0,C 180,E1 -19282.183,E2 -19282.183} C_VEL
LIN {X 0,Y 241.988,Z 746.339,A -85,B 0,C 180,E1 -19285.826,E2 -19285.826} C_VEL
LIN {X 0,Y 241.97,Z 746.345,A -85,B 0,C 180,E1 -19289.589,E2 -19289.589} C_VEL
LIN {X 0,Y 241.98,Z 746.342,A -85,B 0,C 180,E1 -19293.493,E2 -19293.493} C_VEL
LIN {X 0,Y 241.965,Z 746.346,A -85,B 0,C 180,E1 -19297.587,E2 -19297.587} C_VEL
LIN {X 0,Y 241.906,Z 746.351,A -85,B 0,C 180,E1 -19301.93,E2 -19301.93} C_VEL
LIN {X 0,Y 241.9,Z 746.351,A -85,B 0,C 180,E1 -19306.58,E2 -19306.58} C_VEL
LIN {X 0,Y 241.976,Z 746.339,A -85,B 0,C 180,E1 -19311.647,E2 -19311.647} C_VEL
LIN {X 0,Y 241.974,Z 746.343,A -85,B 0,C 180,E1 -19314.487,E2 -19314.487} C_VEL
LIN {X 0,Y 241.95,Z 746.345,A -85,B 0,C 180,E1 -19318.476,E2 -19318.476} C_VEL
LIN {X 0,Y 241.952,Z 746.347,A -85,B 0,C 180,E1 -19322.306,E2 -19322.306} C_VEL
LIN {X 0,Y 241.984,Z 746.341,A -85,B 0,C 180,E1 -19326.008,E2 -19326.008} C_VEL
LIN {X 0,Y 242.02,Z 746.334,A -85,B 0,C 180,E1 -19329.607,E2 -19329.607} C_VEL
LIN {X 0,Y 242.118,Z 746.324,A -85,B 0,C 180,E1 -19333.316,E2 -19333.316} C_VEL
LIN {X 0,Y 242.167,Z 746.316,A -85,B 0,C 180,E1 -19338.279,E2 -19338.279} C_VEL
LIN {X 0,Y 242.374,Z 746.292,A -85,B 0,C 180,E1 -19341.664,E2 -19341.664} C_VEL
LIN {X 0,Y 242.398,Z 746.289,A -85,B 0,C 180,E1 -19343.34,E2 -19343.34} C_VEL
LIN {X 0,Y 242.621,Z 746.26,A -85,B 0,C 180,E1 -19348.34,E2 -19348.34} C_VEL
LIN {X 0,Y 242.62,Z 746.261,A -85,B 0,C 180,E1 -19351.66,E2 -19351.66} C_VEL
LIN {X 0,Y 242.4,Z 746.288,A -85,B 0,C 180,E1 -19356.66,E2 -19356.66} C_VEL
LIN {X 0,Y 242.269,Z 746.305,A -85,B 0,C 180,E1 -19360.024,E2 -19360.024} C_VEL
LIN {X 0,Y 242.17,Z 746.317,A -85,B 0,C 180,E1 -19365.141,E2 -19365.141} C_VEL
LIN {X 0,Y 242.075,Z 746.328,A -85,B 0,C 180,E1 -19368.624,E2 -19368.624} C_VEL
LIN {X 0,Y 242.007,Z 746.339,A -85,B 0,C 180,E1 -19372.181,E2 -19372.181} C_VEL
LIN {X 0,Y 242.035,Z 746.337,A -85,B 0,C 180,E1 -19375.821,E2 -19375.821} C_VEL
LIN {X 0,Y 241.971,Z 746.344,A -85,B 0,C 180,E1 -19379.588,E2 -19379.588} C_VEL
LIN {X 0,Y 241.983,Z 746.341,A -85,B 0,C 180,E1 -19383.493,E2 -19383.493} C_VEL
LIN {X 0,Y 242.045,Z 746.441,A -85,B 0,C 180,E1 -19387.376,E2 -19387.376} C_VEL
LIN {X 0,Y 245.84,Z 759.044,A -85,B 0,C 180,E1 -19388.972,E2 -19388.972} C_VEL
LIN {X 0,Y 249.042,Z 770.749,A -85,B 0,C 180,E1 -19390.738,E2 -19390.738} C_VEL
LIN {X 0,Y 249.648,Z 773.195,A -85,B 0,C 180,E1 -19391.151,E2 -19391.151} C_VEL
LIN {X 0,Y 248.594,Z 784.435,A -85,B 0,C 180,E1 -19392.986,E2 -19392.986} C_VEL
LIN {X 0,Y 247.101,Z 795.008,A -85,B 0,C 180,E1 -19395.111,E2 -19395.111} C_VEL
LIN {X 0,Y 245.705,Z 804.898,A -85,B 0,C 180,E1 -19397.576,E2 -19397.576} C_VEL
LIN {X 0,Y 244.494,Z 813.386,A -85,B 0,C 180,E1 -19400.239,E2 -19400.239} C_VEL
LIN {X 0,Y 243.618,Z 819.728,A -85,B 0,C 180,E1 -19402.712,E2 -19402.712} C_VEL
LIN {X 0,Y 243.058,Z 825.638,A -85,B 0,C 180,E1 -19405.678,E2 -19405.678} C_VEL
LIN {X 0,Y 242.703,Z 829.951,A -85,B 0,C 180,E1 -19408.585,E2 -19408.585} C_VEL
LIN {X 0,Y 242.665,Z 832.071,A -85,B 0,C 180,E1 -19410.505,E2 -19410.505} C_VEL
LIN {X 0,Y 243.021,Z 834.332,A -85,B 0,C 180,E1 -19413.702,E2 -19413.702} C_VEL
LIN {X 0,Y 243.971,Z 835.139,A -85,B 0,C 180,E1 -19417.194,E2 -19417.194} C_VEL
LIN {X 0,Y 245.571,Z 834.103,A -85,B 0,C 180,E1 -19420.81,E2 -19420.81} C_VEL
LIN {X 0,Y 247.11,Z 832.068,A -85,B 0,C 180,E1 -19423.476,E2 -19423.476} C_VEL
LIN {X 0,Y 249.07,Z 828.874,A -85,B 0,C 180,E1 -19426.122,E2 -19426.122} C_VEL
LIN {X 0,Y 251.425,Z 824.448,A -85,B 0,C 180,E1 -19428.716,E2 -19428.716} C_VEL
LIN {X 0,Y 254.158,Z 818.678,A -85,B 0,C 180,E1 -19431.252,E2 -19431.252} C_VEL
LIN {X 0,Y 257.158,Z 811.431,A -85,B 0,C 180,E1 -19433.724,E2 -19433.724} C_VEL
LIN {X 0,Y 260.318,Z 802.974,A -85,B 0,C 180,E1 -19435.965,E2 -19435.965} C_VEL
LIN {X 0,Y 263.122,Z 794.096,A -85,B 0,C 180,E1 -19437.869,E2 -19437.869} C_VEL
LIN {X 0,Y 262.786,Z 790.289,A -85,B 0,C 180,E1 -19438.889,E2 -19438.889} C_VEL
LIN {X 0,Y 260.641,Z 780.735,A -85,B 0,C 180,E1 -19441.545,E2 -19441.545} C_VEL
LIN {X 0,Y 258.307,Z 773.786,A -85,B 0,C 180,E1 -19443.525,E2 -19443.525} C_VEL
LIN {X 0,Y 253.909,Z 764.841,A -85,B 0,C 180,E1 -19446.356,E2 -19446.356} C_VEL
LIN {X 0,Y 249.199,Z 756.522,A -85,B 0,C 180,E1 -19449.216,E2 -19449.216} C_VEL
LIN {X 0,Y 246.845,Z 753.733,A -85,B 0,C 180,E1 -19450.509,E2 -19450.509} C_VEL
LIN {X 0,Y 246.196,Z 752.662,A -85,B 0,C 180,E1 -19450.901,E2 -19450.901} C_VEL
LIN {X 0,Y 243.694,Z 750.614,A -85,B 0,C 180,E1 -19452.264,E2 -19452.264} C_VEL
LIN {X 0,Y 242.741,Z 748.782,A -85,B 0,C 180,E1 -19452.982,E2 -19452.982} C_VEL
LIN {X 0,Y 242.861,Z 749.495,A -85,B 0,C 180,E1 -19457.259,E2 -19457.259} C_VEL
LIN {X 0,Y 243.113,Z 751.001,A -85,B 0,C 180,E1 -19462.074,E2 -19462.074} C_VEL
LIN {X 0,Y 243.624,Z 753.161,A -85,B 0,C 180,E1 -19466.583,E2 -19466.583} C_VEL
LIN {X 0,Y 244.116,Z 755.518,A -85,B 0,C 180,E1 -19470.266,E2 -19470.266} C_VEL
LIN {X 0,Y 244.698,Z 758.095,A -85,B 0,C 180,E1 -19473.6,E2 -19473.6} C_VEL
LIN {X 0,Y 245.593,Z 762.185,A -85,B 0,C 180,E1 -19477.97,E2 -19477.97} C_VEL
LIN {X 0,Y 246.524,Z 766.781,A -85,B 0,C 180,E1 -19482.075,E2 -19482.075} C_VEL
LIN {X 0,Y 246.089,Z 768.036,A -85,B 0,C 180,E1 -19482.942,E2 -19482.942} C_VEL
LIN {X 0,Y 243.639,Z 770.565,A -85,B 0,C 180,E1 -19484.281,E2 -19484.281} C_VEL
LIN {X 0,Y 241.145,Z 773.163,A -85,B 0,C 180,E1 -19485.642,E2 -19485.642} C_VEL
LIN {X 0,Y 240.684,Z 774.534,A -85,B 0,C 180,E1 -19486.532,E2 -19486.532} C_VEL
LIN {X 0,Y 241.174,Z 777.192,A -85,B 0,C 180,E1 -19488.305,E2 -19488.305} C_VEL
LIN {X 0,Y 243.01,Z 782.125,A -85,B 0,C 180,E1 -19489.527,E2 -19489.527} C_VEL
LIN {X 0,Y 243.953,Z 784.396,A -85,B 0,C 180,E1 -19490.128,E2 -19490.128} C_VEL
LIN {X 0,Y 245.152,Z 789.316,A -85,B 0,C 180,E1 -19491.068,E2 -19491.068} C_VEL
LIN {X 0,Y 247.245,Z 800.422,A -85,B 0,C 180,E1 -19493.096,E2 -19493.096} C_VEL
LIN {X 0,Y 248.817,Z 812.666,A -85,B 0,C 180,E1 -19495.222,E2 -19495.222} C_VEL
LIN {X 0,Y 249.326,Z 824.909,A -85,B 0,C 180,E1 -19497.32,E2 -19497.32} C_VEL
LIN {X 0,Y 248.821,Z 836.891,A -85,B 0,C 180,E1 -19499.441,E2 -19499.441} C_VEL
LIN {X 0,Y 247.36,Z 847.78,A -85,B 0,C 180,E1 -19501.521,E2 -19501.521} C_VEL
LIN {X 0,Y 244.677,Z 859.492,A -85,B 0,C 180,E1 -19504.021,E2 -19504.021} C_VEL
LIN {X 0,Y 242.266,Z 868.946,A -85,B 0,C 180,E1 -19506.491,E2 -19506.491} C_VEL
LIN {X 0,Y 239.421,Z 876.868,A -85,B 0,C 180,E1 -19508.925,E2 -19508.925} C_VEL
LIN {X 0,Y 236.776,Z 884.321,A -85,B 0,C 180,E1 -19511.774,E2 -19511.774} C_VEL
LIN {X 0,Y 235.259,Z 889.741,A -85,B 0,C 180,E1 -19514.403,E2 -19514.403} C_VEL
LIN {X 0,Y 234.241,Z 893.988,A -85,B 0,C 180,E1 -19516.995,E2 -19516.995} C_VEL
LIN {X 0,Y 233.749,Z 897.307,A -85,B 0,C 180,E1 -19519.607,E2 -19519.607} C_VEL
LIN {X 0,Y 233.857,Z 900.363,A -85,B 0,C 180,E1 -19523.096,E2 -19523.096} C_VEL
LIN {X 0,Y 234.11,Z 901.271,A -85,B 0,C 180,E1 -19524.833,E2 -19524.833} C_VEL
LIN {X 0,Y 234.39,Z 901.758,A -85,B 0,C 180,E1 -19526.562,E2 -19526.562} C_VEL
LIN {X 0,Y 234.71,Z 901.839,A -85,B 0,C 180,E1 -19528.284,E2 -19528.284} C_VEL
LIN {X 0,Y 235.156,Z 901.52,A -85,B 0,C 180,E1 -19530,E2 -19530} C_VEL
LIN {X 0,Y 234.944,Z 900.646,A -85,B 0,C 180,E1 -19531.714,E2 -19531.714} C_VEL
LIN {X 0,Y 234.696,Z 899.268,A -85,B 0,C 180,E1 -19533.433,E2 -19533.433} C_VEL
LIN {X 0,Y 234.515,Z 896.359,A -85,B 0,C 180,E1 -19536.021,E2 -19536.021} C_VEL
LIN {X 0,Y 234.264,Z 892.251,A -85,B 0,C 180,E1 -19538.627,E2 -19538.627} C_VEL
LIN {X 0,Y 234.447,Z 885.918,A -85,B 0,C 180,E1 -19541.674,E2 -19541.674} C_VEL
LIN {X 0,Y 235.165,Z 878.971,A -85,B 0,C 180,E1 -19544.274,E2 -19544.274} C_VEL
LIN {X 0,Y 236.295,Z 870.273,A -85,B 0,C 180,E1 -19546.857,E2 -19546.857} C_VEL
LIN {X 0,Y 237.648,Z 861.428,A -85,B 0,C 180,E1 -19548.984,E2 -19548.984} C_VEL
LIN {X 0,Y 237.966,Z 857.243,A -85,B 0,C 180,E1 -19549.855,E2 -19549.855} C_VEL
LIN {X 0,Y 237.984,Z 845.988,A -85,B 0,C 180,E1 -19551.89,E2 -19551.89} C_VEL
LIN {X 0,Y 237.763,Z 834.307,A -85,B 0,C 180,E1 -19553.605,E2 -19553.605} C_VEL
LIN {X 0,Y 237.27,Z 821.847,A -85,B 0,C 180,E1 -19555.083,E2 -19555.083} C_VEL
LIN {X 0,Y 236.471,Z 808.165,A -85,B 0,C 180,E1 -19556.326,E2 -19556.326} C_VEL
LIN {X 0,Y 235.51,Z 794.93,A -85,B 0,C 180,E1 -19557.22,E2 -19557.22} C_VEL
LIN {X 0,Y 237.123,Z 785.2,A -85,B 0,C 180,E1 -19562.242,E2 -19562.242} C_VEL
LIN {X 0,Y 239.318,Z 774.948,A -85,B 0,C 180,E1 -19567.542,E2 -19567.542} C_VEL
LIN {X 0,Y 239.634,Z 771.009,A -85,B 0,C 180,E1 -19569.634,E2 -19569.634} C_VEL
LIN {X 0,Y 238.617,Z 765.68,A -85,B 0,C 180,E1 -19572.642,E2 -19572.642} C_VEL
LIN {X 0,Y 237.051,Z 758.224,A -85,B 0,C 180,E1 -19577.008,E2 -19577.008} C_VEL
LIN {X 0,Y 235.786,Z 751.368,A -85,B 0,C 180,E1 -19581.249,E2 -19581.249} C_VEL
LIN {X 0,Y 234.969,Z 747.214,A -85,B 0,C 180,E1 -19584.003,E2 -19584.003} C_VEL
LIN {X 0,Y 234.959,Z 747.217,A -85,B 0,C 180,E1 -19587.425,E2 -19587.425} C_VEL
LIN {X 0,Y 234.952,Z 747.216,A -85,B 0,C 180,E1 -19591.406,E2 -19591.406} C_VEL
LIN {X 0,Y 234.979,Z 747.212,A -85,B 0,C 180,E1 -19595.246,E2 -19595.246} C_VEL
LIN {X 0,Y 235,Z 747.21,A -85,B 0,C 180,E1 -19598.969,E2 -19598.969} C_VEL
LIN {X 0,Y 235.098,Z 747.196,A -85,B 0,C 180,E1 -19603.059,E2 -19603.059} C_VEL
LIN {X 0,Y 235.117,Z 747.197,A -85,B 0,C 180,E1 -19607.922,E2 -19607.922} C_VEL
LIN {X 0,Y 235.333,Z 747.167,A -85,B 0,C 180,E1 -19611.413,E2 -19611.413} C_VEL
LIN {X 0,Y 235.374,Z 747.164,A -85,B 0,C 180,E1 -19613.141,E2 -19613.141} C_VEL
LIN {X 0,Y 235.593,Z 747.137,A -85,B 0,C 180,E1 -19618.291,E2 -19618.291} C_VEL
LIN {X 0,Y 235.594,Z 747.135,A -85,B 0,C 180,E1 -19621.71,E2 -19621.71} C_VEL
LIN {X 0,Y 235.353,Z 747.167,A -85,B 0,C 180,E1 -19626.86,E2 -19626.86} C_VEL
LIN {X 0,Y 235.213,Z 747.183,A -85,B 0,C 180,E1 -19630.328,E2 -19630.328} C_VEL
LIN {X 0,Y 235.087,Z 747.197,A -85,B 0,C 180,E1 -19635.608,E2 -19635.608} C_VEL
LIN {X 0,Y 234.99,Z 747.215,A -85,B 0,C 180,E1 -19639.207,E2 -19639.207} C_VEL
LIN {X 0,Y 234.918,Z 747.221,A -85,B 0,C 180,E1 -19642.888,E2 -19642.888} C_VEL
LIN {X 0,Y 234.927,Z 747.218,A -85,B 0,C 180,E1 -19646.663,E2 -19646.663} C_VEL
LIN {X 0,Y 234.9,Z 747.222,A -85,B 0,C 180,E1 -19650.573,E2 -19650.573} C_VEL
LIN {X 0,Y 234.923,Z 747.217,A -85,B 0,C 180,E1 -19654.64,E2 -19654.64} C_VEL
LIN {X 0,Y 234.913,Z 747.221,A -85,B 0,C 180,E1 -19658.935,E2 -19658.935} C_VEL
LIN {X 0,Y 234.853,Z 747.227,A -85,B 0,C 180,E1 -19663.494,E2 -19663.494} C_VEL
LIN {X 0,Y 234.853,Z 747.229,A -85,B 0,C 180,E1 -19666.506,E2 -19666.506} C_VEL
LIN {X 0,Y 234.919,Z 747.217,A -85,B 0,C 180,E1 -19671.079,E2 -19671.079} C_VEL
LIN {X 0,Y 234.923,Z 747.22,A -85,B 0,C 180,E1 -19675.361,E2 -19675.361} C_VEL
LIN {X 0,Y 234.896,Z 747.22,A -85,B 0,C 180,E1 -19679.427,E2 -19679.427} C_VEL
LIN {X 0,Y 234.941,Z 747.218,A -85,B 0,C 180,E1 -19683.822,E2 -19683.822} C_VEL
LIN {X 0,Y 234.987,Z 747.212,A -85,B 0,C 180,E1 -19688.968,E2 -19688.968} C_VEL
LIN {X 0,Y 235.058,Z 747.204,A -85,B 0,C 180,E1 -19693.092,E2 -19693.092} C_VEL
LIN {X 0,Y 235.099,Z 747.195,A -85,B 0,C 180,E1 -19697.921,E2 -19697.921} C_VEL
LIN {X 0,Y 235.314,Z 747.172,A -85,B 0,C 180,E1 -19701.412,E2 -19701.412} C_VEL
LIN {X 0,Y 235.35,Z 747.168,A -85,B 0,C 180,E1 -19703.14,E2 -19703.14} C_VEL
LIN {X 0,Y 235.58,Z 747.137,A -85,B 0,C 180,E1 -19708.291,E2 -19708.291} C_VEL
LIN {X 0,Y 235.579,Z 747.138,A -85,B 0,C 180,E1 -19711.71,E2 -19711.71} C_VEL
LIN {X 0,Y 235.351,Z 747.166,A -85,B 0,C 180,E1 -19716.86,E2 -19716.86} C_VEL
LIN {X 0,Y 235.216,Z 747.182,A -85,B 0,C 180,E1 -19720.328,E2 -19720.328} C_VEL
LIN {X 0,Y 235.117,Z 747.199,A -85,B 0,C 180,E1 -19725.606,E2 -19725.606} C_VEL
LIN {X 0,Y 235.01,Z 747.21,A -85,B 0,C 180,E1 -19729.206,E2 -19729.206} C_VEL
LIN {X 0,Y 234.949,Z 747.216,A -85,B 0,C 180,E1 -19732.884,E2 -19732.884} C_VEL
LIN {X 0,Y 234.948,Z 747.217,A -85,B 0,C 180,E1 -19736.66,E2 -19736.66} C_VEL
LIN {X 0,Y 234.901,Z 747.224,A -85,B 0,C 180,E1 -19740.572,E2 -19740.572} C_VEL
LIN {X 0,Y 234.937,Z 747.22,A -85,B 0,C 180,E1 -19744.637,E2 -19744.637} C_VEL
LIN {X 0,Y 234.982,Z 747.226,A -85,B 0,C 180,E1 -19746.873,E2 -19746.873} C_VEL
LIN {X 0,Y 238.626,Z 759.238,A -85,B 0,C 180,E1 -19748.433,E2 -19748.433} C_VEL
LIN {X 0,Y 241.729,Z 770.411,A -85,B 0,C 180,E1 -19750.152,E2 -19750.152} C_VEL
LIN {X 0,Y 242.768,Z 775.227,A -85,B 0,C 180,E1 -19750.968,E2 -19750.968} C_VEL
LIN {X 0,Y 241.581,Z 785.777,A -85,B 0,C 180,E1 -19752.754,E2 -19752.754} C_VEL
LIN {X 0,Y 240.067,Z 796.341,A -85,B 0,C 180,E1 -19754.947,E2 -19754.947} C_VEL
LIN {X 0,Y 238.705,Z 805.879,A -85,B 0,C 180,E1 -19757.397,E2 -19757.397} C_VEL
LIN {X 0,Y 237.531,Z 813.884,A -85,B 0,C 180,E1 -19759.956,E2 -19759.956} C_VEL
LIN {X 0,Y 236.622,Z 820.293,A -85,B 0,C 180,E1 -19762.492,E2 -19762.492} C_VEL
LIN {X 0,Y 236.18,Z 824.509,A -85,B 0,C 180,E1 -19764.531,E2 -19764.531} C_VEL
LIN {X 0,Y 235.737,Z 829.447,A -85,B 0,C 180,E1 -19767.545,E2 -19767.545} C_VEL
LIN {X 0,Y 235.601,Z 832.312,A -85,B 0,C 180,E1 -19769.892,E2 -19769.892} C_VEL
LIN {X 0,Y 235.68,Z 833.825,A -85,B 0,C 180,E1 -19771.502,E2 -19771.502} C_VEL
LIN {X 0,Y 235.958,Z 835.178,A -85,B 0,C 180,E1 -19773.463,E2 -19773.463} C_VEL
LIN {X 0,Y 236.844,Z 836.258,A -85,B 0,C 180,E1 -19776.91,E2 -19776.91} C_VEL
LIN {X 0,Y 237.766,Z 836.073,A -85,B 0,C 180,E1 -19779.225,E2 -19779.225} C_VEL
LIN {X 0,Y 238.698,Z 835.399,A -85,B 0,C 180,E1 -19781.102,E2 -19781.102} C_VEL
LIN {X 0,Y 239.764,Z 834.23,A -85,B 0,C 180,E1 -19782.955,E2 -19782.955} C_VEL
LIN {X 0,Y 241.728,Z 831.525,A -85,B 0,C 180,E1 -19785.692,E2 -19785.692} C_VEL
LIN {X 0,Y 244.033,Z 827.655,A -85,B 0,C 180,E1 -19788.369,E2 -19788.369} C_VEL
LIN {X 0,Y 246.814,Z 822.515,A -85,B 0,C 180,E1 -19790.989,E2 -19790.989} C_VEL
LIN {X 0,Y 249.922,Z 815.939,A -85,B 0,C 180,E1 -19793.541,E2 -19793.541} C_VEL
LIN {X 0,Y 253.122,Z 808.165,A -85,B 0,C 180,E1 -19795.885,E2 -19795.885} C_VEL
LIN {X 0,Y 256.382,Z 799.216,A -85,B 0,C 180,E1 -19798.036,E2 -19798.036} C_VEL
LIN {X 0,Y 257.035,Z 797.269,A -85,B 0,C 180,E1 -19798.433,E2 -19798.433} C_VEL
LIN {X 0,Y 257.253,Z 795.285,A -85,B 0,C 180,E1 -19798.947,E2 -19798.947} C_VEL
LIN {X 0,Y 255.911,Z 787.911,A -85,B 0,C 180,E1 -19801.18,E2 -19801.18} C_VEL
LIN {X 0,Y 254.318,Z 781.157,A -85,B 0,C 180,E1 -19803.168,E2 -19803.168} C_VEL
LIN {X 0,Y 251.644,Z 774.408,A -85,B 0,C 180,E1 -19805.358,E2 -19805.358} C_VEL
LIN {X 0,Y 247.038,Z 765.138,A -85,B 0,C 180,E1 -19808.669,E2 -19808.669} C_VEL
LIN {X 0,Y 245.253,Z 761.99,A -85,B 0,C 180,E1 -19809.9,E2 -19809.9} C_VEL
LIN {X 0,Y 243.456,Z 759.531,A -85,B 0,C 180,E1 -19811.036,E2 -19811.036} C_VEL
LIN {X 0,Y 240.263,Z 755.938,A -85,B 0,C 180,E1 -19813.103,E2 -19813.103} C_VEL
LIN {X 0,Y 239.972,Z 755.343,A -85,B 0,C 180,E1 -19813.334,E2 -19813.334} C_VEL
LIN {X 0,Y 237.53,Z 753.827,A -85,B 0,C 180,E1 -19814.894,E2 -19814.894} C_VEL
LIN {X 0,Y 236.137,Z 751.581,A -85,B 0,C 180,E1 -19816.091,E2 -19816.091} C_VEL
LIN {X 0,Y 236.349,Z 752.959,A -85,B 0,C 180,E1 -19820.905,E2 -19820.905} C_VEL
LIN {X 0,Y 236.909,Z 755.443,A -85,B 0,C 180,E1 -19826.422,E2 -19826.422} C_VEL
LIN {X 0,Y 237.504,Z 758.278,A -85,B 0,C 180,E1 -19830.891,E2 -19830.891} C_VEL
LIN {X 0,Y 238.058,Z 760.921,A -85,B 0,C 180,E1 -19834.246,E2 -19834.246} C_VEL
LIN {X 0,Y 239.147,Z 765.624,A -85,B 0,C 180,E1 -19839.177,E2 -19839.177} C_VEL
LIN {X 0,Y 240.089,Z 770.698,A -85,B 0,C 180,E1 -19843.606,E2 -19843.606} C_VEL
LIN {X 0,Y 240.684,Z 774.534,A -85,B 0,C 180,E1 -19846.532,E2 -19846.532} C_VEL
LIN {X 0,Y 240.894,Z 776.23,A -85,B 0,C 180,E1 -19847.362,E2 -19847.362} C_VEL
LIN {X 0,Y 241.094,Z 778.694,A -85,B 0,C 180,E1 -19848.081,E2 -19848.081} C_VEL
LIN {X 0,Y 241.254,Z 781.68,A -85,B 0,C 180,E1 -19848.703,E2 -19848.703} C_VEL
LIN {X 0,Y 241.343,Z 784.959,A -85,B 0,C 180,E1 -19849.24,E2 -19849.24} C_VEL
LIN {X 0,Y 241.535,Z 795.827,A -85,B 0,C 180,E1 -19850.738,E2 -19850.738} C_VEL
LIN {X 0,Y 241.775,Z 799.257,A -85,B 0,C 180,E1 -19851.301,E2 -19851.301} C_VEL
LIN {X 0,Y 243.32,Z 813.36,A -85,B 0,C 180,E1 -19853.974,E2 -19853.974} C_VEL
LIN {X 0,Y 243.648,Z 824.66,A -85,B 0,C 180,E1 -19856.048,E2 -19856.048} C_VEL
LIN {X 0,Y 242.954,Z 836.898,A -85,B 0,C 180,E1 -19858.364,E2 -19858.364} C_VEL
LIN {X 0,Y 241.146,Z 848.702,A -85,B 0,C 180,E1 -19860.74,E2 -19860.74} C_VEL
LIN {X 0,Y 238.282,Z 859.789,A -85,B 0,C 180,E1 -19863.269,E2 -19863.269} C_VEL
LIN {X 0,Y 235.698,Z 868.987,A -85,B 0,C 180,E1 -19865.795,E2 -19865.795} C_VEL
LIN {X 0,Y 233.287,Z 875.489,A -85,B 0,C 180,E1 -19867.878,E2 -19867.878} C_VEL
LIN {X 0,Y 230.702,Z 882.074,A -85,B 0,C 180,E1 -19870.421,E2 -19870.421} C_VEL
LIN {X 0,Y 229.255,Z 885.846,A -85,B 0,C 180,E1 -19872.148,E2 -19872.148} C_VEL
LIN {X 0,Y 227.956,Z 890.638,A -85,B 0,C 180,E1 -19874.807,E2 -19874.807} C_VEL
LIN {X 0,Y 227.014,Z 894.435,A -85,B 0,C 180,E1 -19877.484,E2 -19877.484} C_VEL
LIN {X 0,Y 226.673,Z 898.135,A -85,B 0,C 180,E1 -19881.082,E2 -19881.082} C_VEL
LIN {X 0,Y 226.777,Z 899.373,A -85,B 0,C 180,E1 -19882.879,E2 -19882.879} C_VEL
LIN {X 0,Y 227.048,Z 900.215,A -85,B 0,C 180,E1 -19884.672,E2 -19884.672} C_VEL
LIN {X 0,Y 227.335,Z 900.652,A -85,B 0,C 180,E1 -19886.455,E2 -19886.455} C_VEL
LIN {X 0,Y 227.678,Z 900.689,A -85,B 0,C 180,E1 -19888.231,E2 -19888.231} C_VEL
LIN {X 0,Y 228.142,Z 900.32,A -85,B 0,C 180,E1 -19890,E2 -19890} C_VEL
LIN {X 0,Y 227.931,Z 899.354,A -85,B 0,C 180,E1 -19891.767,E2 -19891.767} C_VEL
LIN {X 0,Y 227.671,Z 897.93,A -85,B 0,C 180,E1 -19893.539,E2 -19893.539} C_VEL
LIN {X 0,Y 227.462,Z 894.912,A -85,B 0,C 180,E1 -19896.208,E2 -19896.208} C_VEL
LIN {X 0,Y 227.228,Z 890.685,A -85,B 0,C 180,E1 -19898.896,E2 -19898.896} C_VEL
LIN {X 0,Y 227.402,Z 885.225,A -85,B 0,C 180,E1 -19901.589,E2 -19901.589} C_VEL
LIN {X 0,Y 228.11,Z 878.391,A -85,B 0,C 180,E1 -19904.269,E2 -19904.269} C_VEL
LIN {X 0,Y 229.227,Z 869.795,A -85,B 0,C 180,E1 -19906.934,E2 -19906.934} C_VEL
LIN {X 0,Y 230.754,Z 860.14,A -85,B 0,C 180,E1 -19909.336,E2 -19909.336} C_VEL
LIN {X 0,Y 230.968,Z 849.854,A -85,B 0,C 180,E1 -19911.416,E2 -19911.416} C_VEL
LIN {X 0,Y 230.852,Z 837.089,A -85,B 0,C 180,E1 -19913.512,E2 -19913.512} C_VEL
LIN {X 0,Y 230.415,Z 825.141,A -85,B 0,C 180,E1 -19915.087,E2 -19915.087} C_VEL
LIN {X 0,Y 229.73,Z 811.148,A -85,B 0,C 180,E1 -19916.516,E2 -19916.516} C_VEL
LIN {X 0,Y 228.829,Z 797.906,A -85,B 0,C 180,E1 -19917.516,E2 -19917.516} C_VEL
LIN {X 0,Y 228.57,Z 793.961,A -85,B 0,C 180,E1 -19917.776,E2 -19917.776} C_VEL
LIN {X 0,Y 230.024,Z 785.437,A -85,B 0,C 180,E1 -19922.322,E2 -19922.322} C_VEL
LIN {X 0,Y 232.079,Z 776.185,A -85,B 0,C 180,E1 -19927.276,E2 -19927.276} C_VEL
LIN {X 0,Y 232.557,Z 773.558,A -85,B 0,C 180,E1 -19928.7,E2 -19928.7} C_VEL
LIN {X 0,Y 232.235,Z 769.762,A -85,B 0,C 180,E1 -19930.838,E2 -19930.838} C_VEL
LIN {X 0,Y 230.597,Z 761.914,A -85,B 0,C 180,E1 -19935.494,E2 -19935.494} C_VEL
LIN {X 0,Y 229.134,Z 754.587,A -85,B 0,C 180,E1 -19940.068,E2 -19940.068} C_VEL
LIN {X 0,Y 227.951,Z 748.088,A -85,B 0,C 180,E1 -19944.413,E2 -19944.413} C_VEL
LIN {X 0,Y 227.91,Z 748.097,A -85,B 0,C 180,E1 -19949.704,E2 -19949.704} C_VEL
LIN {X 0,Y 227.926,Z 748.091,A -85,B 0,C 180,E1 -19954.426,E2 -19954.426} C_VEL
LIN {X 0,Y 227.949,Z 748.091,A -85,B 0,C 180,E1 -19958.286,E2 -19958.286} C_VEL
LIN {X 0,Y 228.036,Z 748.077,A -85,B 0,C 180,E1 -19962.826,E2 -19962.826} C_VEL
LIN {X 0,Y 228.075,Z 748.073,A -85,B 0,C 180,E1 -19967.543,E2 -19967.543} C_VEL
LIN {X 0,Y 228.269,Z 748.047,A -85,B 0,C 180,E1 -19971.145,E2 -19971.145} C_VEL
LIN {X 0,Y 228.325,Z 748.043,A -85,B 0,C 180,E1 -19972.928,E2 -19972.928} C_VEL
LIN {X 0,Y 228.551,Z 748.013,A -85,B 0,C 180,E1 -19978.238,E2 -19978.238} C_VEL
LIN {X 0,Y 228.553,Z 748.013,A -85,B 0,C 180,E1 -19981.762,E2 -19981.762} C_VEL
LIN {X 0,Y 228.305,Z 748.043,A -85,B 0,C 180,E1 -19987.073,E2 -19987.073} C_VEL
LIN {X 0,Y 228.144,Z 748.065,A -85,B 0,C 180,E1 -19990.652,E2 -19990.652} C_VEL
LIN {X 0,Y 228.043,Z 748.076,A -85,B 0,C 180,E1 -19994.274,E2 -19994.274} C_VEL
LIN {X 0,Y 227.97,Z 748.085,A -85,B 0,C 180,E1 -19997.956,E2 -19997.956} C_VEL
LIN {X 0,Y 227.905,Z 748.093,A -85,B 0,C 180,E1 -20002.313,E2 -20002.313} C_VEL
LIN {X 0,Y 227.904,Z 748.092,A -85,B 0,C 180,E1 -20006.583,E2 -20006.583} C_VEL
LIN {X 0,Y 227.875,Z 748.098,A -85,B 0,C 180,E1 -20010.281,E2 -20010.281} C_VEL
LIN {X 0,Y 227.877,Z 748.098,A -85,B 0,C 180,E1 -20013.721,E2 -20013.721} C_VEL
LIN {X 0,Y 227.838,Z 748.104,A -85,B 0,C 180,E1 -20018.093,E2 -20018.093} C_VEL
LIN {X 0,Y 227.785,Z 748.106,A -85,B 0,C 180,E1 -20022.749,E2 -20022.749} C_VEL
LIN {X 0,Y 227.811,Z 748.105,A -85,B 0,C 180,E1 -20025.199,E2 -20025.199} C_VEL
LIN {X 0,Y 227.798,Z 748.108,A -85,B 0,C 180,E1 -20029.617,E2 -20029.617} C_VEL
LIN {X 0,Y 227.863,Z 748.102,A -85,B 0,C 180,E1 -20034.125,E2 -20034.125} C_VEL
LIN {X 0,Y 227.855,Z 748.101,A -85,B 0,C 180,E1 -20038.376,E2 -20038.376} C_VEL
LIN {X 0,Y 227.834,Z 748.106,A -85,B 0,C 180,E1 -20042.438,E2 -20042.438} C_VEL
LIN {X 0,Y 227.871,Z 748.101,A -85,B 0,C 180,E1 -20046.363,E2 -20046.363} C_VEL
LIN {X 0,Y 227.923,Z 748.091,A -85,B 0,C 180,E1 -20050.173,E2 -20050.173} C_VEL
LIN {X 0,Y 228.025,Z 748.079,A -85,B 0,C 180,E1 -20053.896,E2 -20053.896} C_VEL
LIN {X 0,Y 228.057,Z 748.073,A -85,B 0,C 180,E1 -20057.542,E2 -20057.542} C_VEL
LIN {X 0,Y 228.255,Z 748.053,A -85,B 0,C 180,E1 -20061.144,E2 -20061.144} C_VEL
LIN {X 0,Y 228.302,Z 748.048,A -85,B 0,C 180,E1 -20062.927,E2 -20062.927} C_VEL
LIN {X 0,Y 228.538,Z 748.014,A -85,B 0,C 180,E1 -20068.238,E2 -20068.238} C_VEL
LIN {X 0,Y 228.538,Z 748.015,A -85,B 0,C 180,E1 -20071.762,E2 -20071.762} C_VEL
LIN {X 0,Y 228.304,Z 748.045,A -85,B 0,C 180,E1 -20077.073,E2 -20077.073} C_VEL
LIN {X 0,Y 228.147,Z 748.063,A -85,B 0,C 180,E1 -20080.651,E2 -20080.651} C_VEL
LIN {X 0,Y 228.066,Z 748.073,A -85,B 0,C 180,E1 -20084.272,E2 -20084.272} C_VEL
LIN {X 0,Y 228.006,Z 748.083,A -85,B 0,C 180,E1 -20087.953,E2 -20087.953} C_VEL
LIN {X 0,Y 227.924,Z 748.093,A -85,B 0,C 180,E1 -20092.324,E2 -20092.324} C_VEL
LIN {X 0,Y 227.925,Z 748.092,A -85,B 0,C 180,E1 -20096.592,E2 -20096.592} C_VEL
LIN {X 0,Y 227.876,Z 748.1,A -85,B 0,C 180,E1 -20100.281,E2 -20100.281} C_VEL
LIN {X 0,Y 227.88,Z 748.1,A -85,B 0,C 180,E1 -20103.72,E2 -20103.72} C_VEL
LIN {X 0,Y 227.95,Z 748.19,A -85,B 0,C 180,E1 -20106.388,E2 -20106.388} C_VEL
LIN {X 0,Y 231.624,Z 760.375,A -85,B 0,C 180,E1 -20108.018,E2 -20108.018} C_VEL
LIN {X 0,Y 234.747,Z 771.566,A -85,B 0,C 180,E1 -20109.788,E2 -20109.788} C_VEL
LIN {X 0,Y 235.885,Z 776.626,A -85,B 0,C 180,E1 -20110.674,E2 -20110.674} C_VEL
LIN {X 0,Y 234.555,Z 787.274,A -85,B 0,C 180,E1 -20112.547,E2 -20112.547} C_VEL
LIN {X 0,Y 232.975,Z 797.951,A -85,B 0,C 180,E1 -20114.853,E2 -20114.853} C_VEL
LIN {X 0,Y 231.763,Z 806.324,A -85,B 0,C 180,E1 -20117.07,E2 -20117.07} C_VEL
LIN {X 0,Y 230.563,Z 814.268,A -85,B 0,C 180,E1 -20119.646,E2 -20119.646} C_VEL
LIN {X 0,Y 229.492,Z 821.958,A -85,B 0,C 180,E1 -20122.772,E2 -20122.772} C_VEL
LIN {X 0,Y 229.035,Z 826.777,A -85,B 0,C 180,E1 -20125.267,E2 -20125.267} C_VEL
LIN {X 0,Y 228.638,Z 831.567,A -85,B 0,C 180,E1 -20128.496,E2 -20128.496} C_VEL
LIN {X 0,Y 228.57,Z 833.835,A -85,B 0,C 180,E1 -20130.53,E2 -20130.53} C_VEL
LIN {X 0,Y 228.825,Z 835.784,A -85,B 0,C 180,E1 -20132.961,E2 -20132.961} C_VEL
LIN {X 0,Y 229.135,Z 836.665,A -85,B 0,C 180,E1 -20134.57,E2 -20134.57} C_VEL
LIN {X 0,Y 229.709,Z 837.318,A -85,B 0,C 180,E1 -20136.616,E2 -20136.616} C_VEL
LIN {X 0,Y 230.441,Z 837.411,A -85,B 0,C 180,E1 -20138.532,E2 -20138.532} C_VEL
LIN {X 0,Y 231.347,Z 837.066,A -85,B 0,C 180,E1 -20140.478,E2 -20140.478} C_VEL
LIN {X 0,Y 232.393,Z 836.193,A -85,B 0,C 180,E1 -20142.397,E2 -20142.397} C_VEL
LIN {X 0,Y 233.624,Z 834.856,A -85,B 0,C 180,E1 -20144.291,E2 -20144.291} C_VEL
LIN {X 0,Y 235.837,Z 831.926,A -85,B 0,C 180,E1 -20147.085,E2 -20147.085} C_VEL
LIN {X 0,Y 238.469,Z 827.786,A -85,B 0,C 180,E1 -20149.815,E2 -20149.815} C_VEL
LIN {X 0,Y 241.593,Z 822.179,A -85,B 0,C 180,E1 -20152.517,E2 -20152.517} C_VEL
LIN {X 0,Y 244.841,Z 815.394,A -85,B 0,C 180,E1 -20155.06,E2 -20155.06} C_VEL
LIN {X 0,Y 247.984,Z 808.287,A -85,B 0,C 180,E1 -20157.157,E2 -20157.157} C_VEL
LIN {X 0,Y 251.242,Z 799.722,A -85,B 0,C 180,E1 -20159.198,E2 -20159.198} C_VEL
LIN {X 0,Y 251.27,Z 797.026,A -85,B 0,C 180,E1 -20160,E2 -20160} C_VEL
LIN {X 0,Y 249.585,Z 786.869,A -85,B 0,C 180,E1 -20163.228,E2 -20163.228} C_VEL
LIN {X 0,Y 247.656,Z 780.879,A -85,B 0,C 180,E1 -20165.277,E2 -20165.277} C_VEL
LIN {X 0,Y 243.551,Z 771.521,A -85,B 0,C 180,E1 -20168.798,E2 -20168.798} C_VEL
LIN {X 0,Y 242.003,Z 768.516,A -85,B 0,C 180,E1 -20170.035,E2 -20170.035} C_VEL
